LIN {X 0,Y 516.274,Z 395.585,A -85,B 0,C 180,E1 -4997.107,E2 -4997.107} C_VEL
LIN {X 0,Y 516.289,Z 396.844,A -85,B 0,C 180,E1 -4998.208,E2 -4998.208} C_VEL
LIN {X 0,Y 518.463,Z 408.41,A -85,B 0,C 180,E1 -4998.579,E2 -4998.579} C_VEL
LIN {X 0,Y 518.178,Z 420.619,A -85,B 0,C 180,E1 -4999.041,E2 -4999.041} C_VEL
LIN {X 0,Y 517.927,Z 432.987,A -85,B 0,C 180,E1 -4999.678,E2 -4999.678} C_VEL
LIN {X 0,Y 517.573,Z 444.529,A -85,B 0,C 180,E1 -5000.457,E2 -5000.457} C_VEL
LIN {X 0,Y 517.31,Z 455.837,A -85,B 0,C 180,E1 -5001.422,E2 -5001.422} C_VEL
LIN {X 0,Y 517.018,Z 465.136,A -85,B 0,C 180,E1 -5002.412,E2 -5002.412} C_VEL
LIN {X 0,Y 516.779,Z 473.686,A -85,B 0,C 180,E1 -5003.535,E2 -5003.535} C_VEL
LIN {X 0,Y 516.539,Z 480.957,A -85,B 0,C 180,E1 -5004.714,E2 -5004.714} C_VEL
LIN {X 0,Y 516.446,Z 486.584,A -85,B 0,C 180,E1 -5005.852,E2 -5005.852} C_VEL
LIN {X 0,Y 516.334,Z 491.147,A -85,B 0,C 180,E1 -5007.014,E2 -5007.014} C_VEL
LIN {X 0,Y 516.286,Z 495.193,A -85,B 0,C 180,E1 -5008.394,E2 -5008.394} C_VEL
LIN {X 0,Y 516.191,Z 497.831,A -85,B 0,C 180,E1 -5009.752,E2 -5009.752} C_VEL
LIN {X 0,Y 516.199,Z 498.912,A -85,B 0,C 180,E1 -5010.651,E2 -5010.651} C_VEL
LIN {X 0,Y 516.184,Z 499.461,A -85,B 0,C 180,E1 -5011.542,E2 -5011.542} C_VEL
LIN {X 0,Y 516.169,Z 499.49,A -85,B 0,C 180,E1 -5012.424,E2 -5012.424} C_VEL
LIN {X 0,Y 516.169,Z 499.058,A -85,B 0,C 180,E1 -5013.301,E2 -5013.301} C_VEL
LIN {X 0,Y 516.186,Z 498.084,A -85,B 0,C 180,E1 -5014.172,E2 -5014.172} C_VEL
LIN {X 0,Y 516.267,Z 496.647,A -85,B 0,C 180,E1 -5015.04,E2 -5015.04} C_VEL
LIN {X 0,Y 516.337,Z 493.561,A -85,B 0,C 180,E1 -5016.327,E2 -5016.327} C_VEL
LIN {X 0,Y 516.436,Z 488.822,A -85,B 0,C 180,E1 -5017.715,E2 -5017.715} C_VEL
LIN {X 0,Y 516.545,Z 482.626,A -85,B 0,C 180,E1 -5019.075,E2 -5019.075} C_VEL
LIN {X 0,Y 516.722,Z 475.326,A -85,B 0,C 180,E1 -5020.329,E2 -5020.329} C_VEL
LIN {X 0,Y 516.922,Z 467.803,A -85,B 0,C 180,E1 -5021.368,E2 -5021.368} C_VEL
LIN {X 0,Y 517.231,Z 458.063,A -85,B 0,C 180,E1 -5022.46,E2 -5022.46} C_VEL
LIN {X 0,Y 517.467,Z 448.555,A -85,B 0,C 180,E1 -5023.328,E2 -5023.328} C_VEL
LIN {X 0,Y 517.786,Z 437.368,A -85,B 0,C 180,E1 -5024.148,E2 -5024.148} C_VEL
LIN {X 0,Y 518.106,Z 425.293,A -85,B 0,C 180,E1 -5024.836,E2 -5024.836} C_VEL
LIN {X 0,Y 518.392,Z 412.692,A -85,B 0,C 180,E1 -5025.375,E2 -5025.375} C_VEL
LIN {X 0,Y 518.315,Z 407.593,A -85,B 0,C 180,E1 -5025.548,E2 -5025.548} C_VEL
LIN {X 0,Y 516.347,Z 397.146,A -85,B 0,C 180,E1 -5025.894,E2 -5025.894} C_VEL
LIN {X 0,Y 516.355,Z 393.731,A -85,B 0,C 180,E1 -5029.016,E2 -5029.016} C_VEL
LIN {X 0,Y 516.424,Z 390.407,A -85,B 0,C 180,E1 -5032.179,E2 -5032.179} C_VEL
LIN {X 0,Y 516.475,Z 387.929,A -85,B 0,C 180,E1 -5034.535,E2 -5034.535} C_VEL
LIN {X 0,Y 516.447,Z 385.452,A -85,B 0,C 180,E1 -5036.88,E2 -5036.88} C_VEL
LIN {X 0,Y 516.657,Z 382.989,A -85,B 0,C 180,E1 -5039.221,E2 -5039.221} C_VEL
LIN {X 0,Y 516.81,Z 381.331,A -85,B 0,C 180,E1 -5040.78,E2 -5040.78} C_VEL
LIN {X 0,Y 516.793,Z 377.272,A -85,B 0,C 180,E1 -5044.681,E2 -5044.681} C_VEL
LIN {X 0,Y 516.754,Z 376.473,A -85,B 0,C 180,E1 -5045.464,E2 -5045.464} C_VEL
LIN {X 0,Y 516.909,Z 376.103,A -85,B 0,C 180,E1 -5047.049,E2 -5047.049} C_VEL
LIN {X 0,Y 516.929,Z 376.095,A -85,B 0,C 180,E1 -5049.39,E2 -5049.39} C_VEL
LIN {X 0,Y 516.965,Z 376.093,A -85,B 0,C 180,E1 -5051.836,E2 -5051.836} C_VEL
LIN {X 0,Y 516.909,Z 376.097,A -85,B 0,C 180,E1 -5055.149,E2 -5055.149} C_VEL
LIN {X 0,Y 516.897,Z 376.098,A -85,B 0,C 180,E1 -5058.224,E2 -5058.224} C_VEL
LIN {X 0,Y 516.883,Z 376.103,A -85,B 0,C 180,E1 -5060.703,E2 -5060.703} C_VEL
LIN {X 0,Y 516.877,Z 376.1,A -85,B 0,C 180,E1 -5063.224,E2 -5063.224} C_VEL
LIN {X 0,Y 516.913,Z 376.096,A -85,B 0,C 180,E1 -5066.199,E2 -5066.199} C_VEL
LIN {X 0,Y 516.912,Z 376.098,A -85,B 0,C 180,E1 -5069.306,E2 -5069.306} C_VEL
LIN {X 0,Y 516.872,Z 376.104,A -85,B 0,C 180,E1 -5072.547,E2 -5072.547} C_VEL
LIN {X 0,Y 516.86,Z 376.106,A -85,B 0,C 180,E1 -5075.336,E2 -5075.336} C_VEL
LIN {X 0,Y 516.86,Z 376.103,A -85,B 0,C 180,E1 -5077.947,E2 -5077.947} C_VEL
LIN {X 0,Y 516.892,Z 376.1,A -85,B 0,C 180,E1 -5080.741,E2 -5080.741} C_VEL
LIN {X 0,Y 516.86,Z 376.104,A -85,B 0,C 180,E1 -5083.906,E2 -5083.906} C_VEL
LIN {X 0,Y 516.861,Z 376.105,A -85,B 0,C 180,E1 -5086.11,E2 -5086.11} C_VEL
LIN {X 0,Y 516.889,Z 376.104,A -85,B 0,C 180,E1 -5089.264,E2 -5089.264} C_VEL
LIN {X 0,Y 516.933,Z 376.22,A -85,B 0,C 180,E1 -5091.051,E2 -5091.051} C_VEL
LIN {X 0,Y 517.978,Z 382.454,A -85,B 0,C 180,E1 -5093.833,E2 -5093.833} C_VEL
LIN {X 0,Y 517.929,Z 387.606,A -85,B 0,C 180,E1 -5095.867,E2 -5095.867} C_VEL
LIN {X 0,Y 517.555,Z 395.985,A -85,B 0,C 180,E1 -5098.939,E2 -5098.939} C_VEL
LIN {X 0,Y 517.232,Z 404.927,A -85,B 0,C 180,E1 -5102.032,E2 -5102.032} C_VEL
LIN {X 0,Y 517.067,Z 414.228,A -85,B 0,C 180,E1 -5105.084,E2 -5105.084} C_VEL
LIN {X 0,Y 516.883,Z 423.643,A -85,B 0,C 180,E1 -5108.047,E2 -5108.047} C_VEL
LIN {X 0,Y 516.771,Z 431.808,A -85,B 0,C 180,E1 -5110.541,E2 -5110.541} C_VEL
LIN {X 0,Y 516.6,Z 441.466,A -85,B 0,C 180,E1 -5113.403,E2 -5113.403} C_VEL
LIN {X 0,Y 516.532,Z 450.706,A -85,B 0,C 180,E1 -5116.103,E2 -5116.103} C_VEL
LIN {X 0,Y 518.459,Z 463.813,A -85,B 0,C 180,E1 -5116.456,E2 -5116.456} C_VEL
LIN {X 0,Y 518.157,Z 476.925,A -85,B 0,C 180,E1 -5116.922,E2 -5116.922} C_VEL
LIN {X 0,Y 517.848,Z 489.403,A -85,B 0,C 180,E1 -5117.537,E2 -5117.537} C_VEL
LIN {X 0,Y 517.538,Z 500.606,A -85,B 0,C 180,E1 -5118.25,E2 -5118.25} C_VEL
LIN {X 0,Y 517.266,Z 511.613,A -85,B 0,C 180,E1 -5119.137,E2 -5119.137} C_VEL
LIN {X 0,Y 516.998,Z 520.585,A -85,B 0,C 180,E1 -5120.022,E2 -5120.022} C_VEL
LIN {X 0,Y 516.746,Z 530.339,A -85,B 0,C 180,E1 -5121.202,E2 -5121.202} C_VEL
LIN {X 0,Y 516.56,Z 538.106,A -85,B 0,C 180,E1 -5122.38,E2 -5122.38} C_VEL
LIN {X 0,Y 516.423,Z 545.262,A -85,B 0,C 180,E1 -5123.753,E2 -5123.753} C_VEL
LIN {X 0,Y 516.313,Z 550.022,A -85,B 0,C 180,E1 -5124.927,E2 -5124.927} C_VEL
LIN {X 0,Y 516.354,Z 553.665,A -85,B 0,C 180,E1 -5126.101,E2 -5126.101} C_VEL
LIN {X 0,Y 516.282,Z 555.538,A -85,B 0,C 180,E1 -5126.882,E2 -5126.882} C_VEL
LIN {X 0,Y 516.261,Z 556.944,A -85,B 0,C 180,E1 -5127.662,E2 -5127.662} C_VEL
LIN {X 0,Y 516.16,Z 558.554,A -85,B 0,C 180,E1 -5129.223,E2 -5129.223} C_VEL
LIN {X 0,Y 516.154,Z 558.771,A -85,B 0,C 180,E1 -5130.003,E2 -5130.003} C_VEL
LIN {X 0,Y 516.192,Z 557.944,A -85,B 0,C 180,E1 -5131.563,E2 -5131.563} C_VEL
LIN {X 0,Y 516.262,Z 556.945,A -85,B 0,C 180,E1 -5132.343,E2 -5132.343} C_VEL
LIN {X 0,Y 516.283,Z 555.54,A -85,B 0,C 180,E1 -5133.124,E2 -5133.124} C_VEL
LIN {X 0,Y 516.327,Z 552.586,A -85,B 0,C 180,E1 -5134.296,E2 -5134.296} C_VEL
LIN {X 0,Y 516.407,Z 548.586,A -85,B 0,C 180,E1 -5135.469,E2 -5135.469} C_VEL
LIN {X 0,Y 516.449,Z 543.248,A -85,B 0,C 180,E1 -5136.683,E2 -5136.683} C_VEL
LIN {X 0,Y 516.582,Z 536.95,A -85,B 0,C 180,E1 -5137.822,E2 -5137.822} C_VEL
LIN {X 0,Y 516.801,Z 528.869,A -85,B 0,C 180,E1 -5139,E2 -5139} C_VEL
LIN {X 0,Y 516.998,Z 520.632,A -85,B 0,C 180,E1 -5139.984,E2 -5139.984} C_VEL
LIN {X 0,Y 517.317,Z 510.597,A -85,B 0,C 180,E1 -5140.967,E2 -5140.967} C_VEL
LIN {X 0,Y 517.57,Z 500.686,A -85,B 0,C 180,E1 -5141.755,E2 -5141.755} C_VEL
LIN {X 0,Y 517.853,Z 489.517,A -85,B 0,C 180,E1 -5142.467,E2 -5142.467} C_VEL
LIN {X 0,Y 518.182,Z 476.997,A -85,B 0,C 180,E1 -5143.084,E2 -5143.084} C_VEL
LIN {X 0,Y 518.44,Z 463.848,A -85,B 0,C 180,E1 -5143.551,E2 -5143.551} C_VEL
LIN {X 0,Y 516.539,Z 450.746,A -85,B 0,C 180,E1 -5143.903,E2 -5143.903} C_VEL
LIN {X 0,Y 516.628,Z 441.751,A -85,B 0,C 180,E1 -5146.602,E2 -5146.602} C_VEL
LIN {X 0,Y 516.807,Z 432.31,A -85,B 0,C 180,E1 -5149.464,E2 -5149.464} C_VEL
LIN {X 0,Y 516.99,Z 421.628,A -85,B 0,C 180,E1 -5152.797,E2 -5152.797} C_VEL
LIN {X 0,Y 517.182,Z 412.366,A -85,B 0,C 180,E1 -5155.778,E2 -5155.778} C_VEL
LIN {X 0,Y 517.425,Z 403.177,A -85,B 0,C 180,E1 -5158.83,E2 -5158.83} C_VEL
LIN {X 0,Y 517.77,Z 394.07,A -85,B 0,C 180,E1 -5161.965,E2 -5161.965} C_VEL
LIN {X 0,Y 518.027,Z 387.92,A -85,B 0,C 180,E1 -5164.149,E2 -5164.149} C_VEL
LIN {X 0,Y 517.995,Z 382.478,A -85,B 0,C 180,E1 -5166.173,E2 -5166.173} C_VEL
LIN {X 0,Y 516.905,Z 376.101,A -85,B 0,C 180,E1 -5168.716,E2 -5168.716} C_VEL
LIN {X 0,Y 516.895,Z 376.102,A -85,B 0,C 180,E1 -5171.779,E2 -5171.779} C_VEL
LIN {X 0,Y 516.908,Z 376.096,A -85,B 0,C 180,E1 -5175.008,E2 -5175.008} C_VEL
LIN {X 0,Y 516.914,Z 376.098,A -85,B 0,C 180,E1 -5178.401,E2 -5178.401} C_VEL
LIN {X 0,Y 516.887,Z 376.103,A -85,B 0,C 180,E1 -5181.284,E2 -5181.284} C_VEL
LIN {X 0,Y 516.878,Z 376.102,A -85,B 0,C 180,E1 -5184.22,E2 -5184.22} C_VEL
LIN {X 0,Y 516.892,Z 376.1,A -85,B 0,C 180,E1 -5187.052,E2 -5187.052} C_VEL
LIN {X 0,Y 516.897,Z 376.098,A -85,B 0,C 180,E1 -5189.796,E2 -5189.796} C_VEL
LIN {X 0,Y 516.9,Z 376.098,A -85,B 0,C 180,E1 -5192.465,E2 -5192.465} C_VEL
LIN {X 0,Y 516.893,Z 376.1,A -85,B 0,C 180,E1 -5195.643,E2 -5195.643} C_VEL
LIN {X 0,Y 516.896,Z 376.099,A -85,B 0,C 180,E1 -5198.462,E2 -5198.462} C_VEL
LIN {X 0,Y 516.909,Z 376.098,A -85,B 0,C 180,E1 -5200.955,E2 -5200.955} C_VEL
LIN {X 0,Y 516.914,Z 376.096,A -85,B 0,C 180,E1 -5203.41,E2 -5203.41} C_VEL
LIN {X 0,Y 516.887,Z 376.099,A -85,B 0,C 180,E1 -5205.833,E2 -5205.833} C_VEL
LIN {X 0,Y 516.977,Z 376.091,A -85,B 0,C 180,E1 -5208.233,E2 -5208.233} C_VEL
LIN {X 0,Y 516.963,Z 376.09,A -85,B 0,C 180,E1 -5211.399,E2 -5211.399} C_VEL
LIN {X 0,Y 516.997,Z 376.086,A -85,B 0,C 180,E1 -5213.756,E2 -5213.756} C_VEL
LIN {X 0,Y 517.019,Z 376.084,A -85,B 0,C 180,E1 -5216.882,E2 -5216.882} C_VEL
LIN {X 0,Y 517.092,Z 376.076,A -85,B 0,C 180,E1 -5219.999,E2 -5219.999} C_VEL
LIN {X 0,Y 517.082,Z 376.075,A -85,B 0,C 180,E1 -5222.336,E2 -5222.336} C_VEL
LIN {X 0,Y 517.022,Z 376.085,A -85,B 0,C 180,E1 -5225.459,E2 -5225.459} C_VEL
LIN {X 0,Y 516.959,Z 376.092,A -85,B 0,C 180,E1 -5228.6,E2 -5228.6} C_VEL
LIN {X 0,Y 516.961,Z 376.09,A -85,B 0,C 180,E1 -5231.806,E2 -5231.806} C_VEL
LIN {X 0,Y 516.95,Z 376.093,A -85,B 0,C 180,E1 -5235.144,E2 -5235.144} C_VEL
LIN {X 0,Y 516.92,Z 376.095,A -85,B 0,C 180,E1 -5238.222,E2 -5238.222} C_VEL
LIN {X 0,Y 516.919,Z 376.097,A -85,B 0,C 180,E1 -5240.7,E2 -5240.7} C_VEL
LIN {X 0,Y 516.896,Z 376.099,A -85,B 0,C 180,E1 -5244.072,E2 -5244.072} C_VEL
LIN {X 0,Y 516.918,Z 376.097,A -85,B 0,C 180,E1 -5246.657,E2 -5246.657} C_VEL
LIN {X 0,Y 516.914,Z 376.098,A -85,B 0,C 180,E1 -5249.522,E2 -5249.522} C_VEL
LIN {X 0,Y 516.901,Z 376.1,A -85,B 0,C 180,E1 -5252.542,E2 -5252.542} C_VEL
LIN {X 0,Y 516.869,Z 376.102,A -85,B 0,C 180,E1 -5255.328,E2 -5255.328} C_VEL
LIN {X 0,Y 516.883,Z 376.102,A -85,B 0,C 180,E1 -5257.941,E2 -5257.941} C_VEL
LIN {X 0,Y 516.886,Z 376.101,A -85,B 0,C 180,E1 -5260.74,E2 -5260.74} C_VEL
LIN {X 0,Y 516.885,Z 376.099,A -85,B 0,C 180,E1 -5263.902,E2 -5263.902} C_VEL
LIN {X 0,Y 516.851,Z 376.104,A -85,B 0,C 180,E1 -5266.894,E2 -5266.894} C_VEL
LIN {X 0,Y 516.887,Z 376.101,A -85,B 0,C 180,E1 -5269.588,E2 -5269.588} C_VEL
LIN {X 0,Y 516.885,Z 376.101,A -85,B 0,C 180,E1 -5270.282,E2 -5270.282} C_VEL
LIN {X 0,Y 516.213,Z 376.186,A -85,B 0,C 180,E1 -5270.932,E2 -5270.932} C_VEL
LIN {X 0,Y 513.368,Z 376.541,A -85,B 0,C 180,E1 -5271.987,E2 -5271.987} C_VEL
LIN {X 0,Y 510.962,Z 376.842,A -85,B 0,C 180,E1 -5272.838,E2 -5272.838} C_VEL
LIN {X 0,Y 509.921,Z 376.969,A -85,B 0,C 180,E1 -5273.494,E2 -5273.494} C_VEL
LIN {X 0,Y 509.832,Z 376.979,A -85,B 0,C 180,E1 -5273.716,E2 -5273.716} C_VEL
LIN {X 0,Y 509.863,Z 376.978,A -85,B 0,C 180,E1 -5276.537,E2 -5276.537} C_VEL
LIN {X 0,Y 509.847,Z 376.978,A -85,B 0,C 180,E1 -5279.332,E2 -5279.332} C_VEL
LIN {X 0,Y 509.887,Z 376.974,A -85,B 0,C 180,E1 -5282.052,E2 -5282.052} C_VEL
LIN {X 0,Y 509.878,Z 376.974,A -85,B 0,C 180,E1 -5284.702,E2 -5284.702} C_VEL
LIN {X 0,Y 509.828,Z 376.981,A -85,B 0,C 180,E1 -5287.455,E2 -5287.455} C_VEL
LIN {X 0,Y 509.916,Z 376.97,A -85,B 0,C 180,E1 -5289.842,E2 -5289.842} C_VEL
LIN {X 0,Y 509.877,Z 376.971,A -85,B 0,C 180,E1 -5293.172,E2 -5293.172} C_VEL
LIN {X 0,Y 509.861,Z 376.976,A -85,B 0,C 180,E1 -5295.632,E2 -5295.632} C_VEL
LIN {X 0,Y 509.911,Z 376.97,A -85,B 0,C 180,E1 -5298.872,E2 -5298.872} C_VEL
LIN {X 0,Y 509.947,Z 376.967,A -85,B 0,C 180,E1 -5302.076,E2 -5302.076} C_VEL
LIN {X 0,Y 509.976,Z 376.963,A -85,B 0,C 180,E1 -5304.461,E2 -5304.461} C_VEL
LIN {X 0,Y 510.051,Z 376.953,A -85,B 0,C 180,E1 -5307.628,E2 -5307.628} C_VEL
LIN {X 0,Y 510.055,Z 376.951,A -85,B 0,C 180,E1 -5310.787,E2 -5310.787} C_VEL
LIN {X 0,Y 509.946,Z 376.964,A -85,B 0,C 180,E1 -5313.157,E2 -5313.157} C_VEL
LIN {X 0,Y 509.974,Z 376.962,A -85,B 0,C 180,E1 -5316.327,E2 -5316.327} C_VEL
LIN {X 0,Y 509.905,Z 376.969,A -85,B 0,C 180,E1 -5318.717,E2 -5318.717} C_VEL
LIN {X 0,Y 509.938,Z 376.967,A -85,B 0,C 180,E1 -5321.927,E2 -5321.927} C_VEL
LIN {X 0,Y 509.878,Z 376.973,A -85,B 0,C 180,E1 -5325.239,E2 -5325.239} C_VEL
LIN {X 0,Y 509.872,Z 376.974,A -85,B 0,C 180,E1 -5327.998,E2 -5327.998} C_VEL
LIN {X 0,Y 509.833,Z 376.978,A -85,B 0,C 180,E1 -5330.999,E2 -5330.999} C_VEL
LIN {X 0,Y 509.84,Z 376.977,A -85,B 0,C 180,E1 -5333.559,E2 -5333.559} C_VEL
LIN {X 0,Y 509.821,Z 376.981,A -85,B 0,C 180,E1 -5336.36,E2 -5336.36} C_VEL
LIN {X 0,Y 509.582,Z 377.013,A -85,B 0,C 180,E1 -5338.858,E2 -5338.858} C_VEL
LIN {X 0,Y 509.456,Z 377.033,A -85,B 0,C 180,E1 -5339.772,E2 -5339.772} C_VEL
LIN {X 0,Y 509.378,Z 380.119,A -85,B 0,C 180,E1 -5342.689,E2 -5342.689} C_VEL
LIN {X 0,Y 509.319,Z 383.194,A -85,B 0,C 180,E1 -5345.5,E2 -5345.5} C_VEL
LIN {X 0,Y 509.284,Z 386.378,A -85,B 0,C 180,E1 -5348.383,E2 -5348.383} C_VEL
LIN {X 0,Y 509.246,Z 389.82,A -85,B 0,C 180,E1 -5351.481,E2 -5351.481} C_VEL
LIN {X 0,Y 509.212,Z 393.462,A -85,B 0,C 180,E1 -5354.734,E2 -5354.734} C_VEL
LIN {X 0,Y 509.216,Z 397.177,A -85,B 0,C 180,E1 -5358.003,E2 -5358.003} C_VEL
LIN {X 0,Y 511.501,Z 409.221,A -85,B 0,C 180,E1 -5358.41,E2 -5358.41} C_VEL
LIN {X 0,Y 511.27,Z 422.157,A -85,B 0,C 180,E1 -5358.92,E2 -5358.92} C_VEL
LIN {X 0,Y 511.011,Z 433.292,A -85,B 0,C 180,E1 -5359.51,E2 -5359.51} C_VEL
LIN {X 0,Y 510.629,Z 445.146,A -85,B 0,C 180,E1 -5360.322,E2 -5360.322} C_VEL
LIN {X 0,Y 510.355,Z 455.392,A -85,B 0,C 180,E1 -5361.204,E2 -5361.204} C_VEL
LIN {X 0,Y 510.057,Z 464.675,A -85,B 0,C 180,E1 -5362.183,E2 -5362.183} C_VEL
LIN {X 0,Y 509.77,Z 473.618,A -85,B 0,C 180,E1 -5363.356,E2 -5363.356} C_VEL
LIN {X 0,Y 509.527,Z 481.237,A -85,B 0,C 180,E1 -5364.599,E2 -5364.599} C_VEL
LIN {X 0,Y 509.373,Z 487.418,A -85,B 0,C 180,E1 -5365.87,E2 -5365.87} C_VEL
LIN {X 0,Y 509.287,Z 491.531,A -85,B 0,C 180,E1 -5366.946,E2 -5366.946} C_VEL
LIN {X 0,Y 509.219,Z 495.639,A -85,B 0,C 180,E1 -5368.369,E2 -5368.369} C_VEL
LIN {X 0,Y 509.147,Z 497.527,A -85,B 0,C 180,E1 -5369.289,E2 -5369.289} C_VEL
LIN {X 0,Y 509.128,Z 499.087,A -85,B 0,C 180,E1 -5370.409,E2 -5370.409} C_VEL
LIN {X 0,Y 509.087,Z 499.965,A -85,B 0,C 180,E1 -5372.007,E2 -5372.007} C_VEL
LIN {X 0,Y 509.087,Z 499.72,A -85,B 0,C 180,E1 -5372.899,E2 -5372.899} C_VEL
LIN {X 0,Y 509.107,Z 498.999,A -85,B 0,C 180,E1 -5373.795,E2 -5373.795} C_VEL
LIN {X 0,Y 509.155,Z 497.809,A -85,B 0,C 180,E1 -5374.667,E2 -5374.667} C_VEL
LIN {X 0,Y 509.244,Z 494.958,A -85,B 0,C 180,E1 -5376.014,E2 -5376.014} C_VEL
LIN {X 0,Y 509.354,Z 491.143,A -85,B 0,C 180,E1 -5377.274,E2 -5377.274} C_VEL
LIN {X 0,Y 509.422,Z 486.001,A -85,B 0,C 180,E1 -5378.557,E2 -5378.557} C_VEL
LIN {X 0,Y 509.631,Z 479.445,A -85,B 0,C 180,E1 -5379.834,E2 -5379.834} C_VEL
LIN {X 0,Y 509.813,Z 472.712,A -85,B 0,C 180,E1 -5380.89,E2 -5380.89} C_VEL
LIN {X 0,Y 510.068,Z 463.686,A -85,B 0,C 180,E1 -5382.038,E2 -5382.038} C_VEL
LIN {X 0,Y 510.389,Z 453.425,A -85,B 0,C 180,E1 -5383.09,E2 -5383.09} C_VEL
LIN {X 0,Y 510.721,Z 443.332,A -85,B 0,C 180,E1 -5383.923,E2 -5383.923} C_VEL
LIN {X 0,Y 511.051,Z 432.035,A -85,B 0,C 180,E1 -5384.664,E2 -5384.664} C_VEL
LIN {X 0,Y 511.352,Z 420.106,A -85,B 0,C 180,E1 -5385.271,E2 -5385.271} C_VEL
LIN {X 0,Y 511.444,Z 408.72,A -85,B 0,C 180,E1 -5385.706,E2 -5385.706} C_VEL
LIN {X 0,Y 509.573,Z 399.17,A -85,B 0,C 180,E1 -5386.021,E2 -5386.021} C_VEL
LIN {X 0,Y 509.261,Z 397.636,A -85,B 0,C 180,E1 -5386.076,E2 -5386.076} C_VEL
LIN {X 0,Y 509.298,Z 394.628,A -85,B 0,C 180,E1 -5388.862,E2 -5388.862} C_VEL
LIN {X 0,Y 509.356,Z 391.228,A -85,B 0,C 180,E1 -5392.07,E2 -5392.07} C_VEL
LIN {X 0,Y 509.409,Z 388.715,A -85,B 0,C 180,E1 -5394.459,E2 -5394.459} C_VEL
LIN {X 0,Y 509.389,Z 386.246,A -85,B 0,C 180,E1 -5396.837,E2 -5396.837} C_VEL
LIN {X 0,Y 509.605,Z 383.758,A -85,B 0,C 180,E1 -5399.211,E2 -5399.211} C_VEL
LIN {X 0,Y 509.771,Z 382.109,A -85,B 0,C 180,E1 -5400.791,E2 -5400.791} C_VEL
LIN {X 0,Y 509.756,Z 378.043,A -85,B 0,C 180,E1 -5404.746,E2 -5404.746} C_VEL
LIN {X 0,Y 509.718,Z 377.23,A -85,B 0,C 180,E1 -5405.539,E2 -5405.539} C_VEL
LIN {X 0,Y 509.883,Z 376.974,A -85,B 0,C 180,E1 -5407.923,E2 -5407.923} C_VEL
LIN {X 0,Y 509.904,Z 376.969,A -85,B 0,C 180,E1 -5411.126,E2 -5411.126} C_VEL
LIN {X 0,Y 509.84,Z 376.979,A -85,B 0,C 180,E1 -5413.553,E2 -5413.553} C_VEL
LIN {X 0,Y 509.836,Z 376.979,A -85,B 0,C 180,E1 -5416.004,E2 -5416.004} C_VEL
LIN {X 0,Y 509.838,Z 376.977,A -85,B 0,C 180,E1 -5418.485,E2 -5418.485} C_VEL
LIN {X 0,Y 509.828,Z 376.98,A -85,B 0,C 180,E1 -5421.003,E2 -5421.003} C_VEL
LIN {X 0,Y 509.835,Z 376.981,A -85,B 0,C 180,E1 -5423.564,E2 -5423.564} C_VEL
LIN {X 0,Y 509.882,Z 376.973,A -85,B 0,C 180,E1 -5426.382,E2 -5426.382} C_VEL
LIN {X 0,Y 509.859,Z 376.974,A -85,B 0,C 180,E1 -5428.846,E2 -5428.846} C_VEL
LIN {X 0,Y 509.796,Z 376.983,A -85,B 0,C 180,E1 -5431.592,E2 -5431.592} C_VEL
LIN {X 0,Y 509.828,Z 376.98,A -85,B 0,C 180,E1 -5434.416,E2 -5434.416} C_VEL
LIN {X 0,Y 509.798,Z 376.984,A -85,B 0,C 180,E1 -5437.343,E2 -5437.343} C_VEL
LIN {X 0,Y 509.854,Z 376.977,A -85,B 0,C 180,E1 -5440.381,E2 -5440.381} C_VEL
LIN {X 0,Y 509.818,Z 376.983,A -85,B 0,C 180,E1 -5443.068,E2 -5443.068} C_VEL
LIN {X 0,Y 509.809,Z 376.984,A -85,B 0,C 180,E1 -5445.796,E2 -5445.796} C_VEL
LIN {X 0,Y 509.851,Z 376.981,A -85,B 0,C 180,E1 -5448.58,E2 -5448.58} C_VEL
LIN {X 0,Y 509.89,Z 377.177,A -85,B 0,C 180,E1 -5450.784,E2 -5450.784} C_VEL
LIN {X 0,Y 511.011,Z 383.665,A -85,B 0,C 180,E1 -5453.75,E2 -5453.75} C_VEL
LIN {X 0,Y 510.963,Z 388.44,A -85,B 0,C 180,E1 -5455.677,E2 -5455.677} C_VEL
LIN {X 0,Y 510.572,Z 396.168,A -85,B 0,C 180,E1 -5458.587,E2 -5458.587} C_VEL
LIN {X 0,Y 510.288,Z 402.199,A -85,B 0,C 180,E1 -5460.734,E2 -5460.734} C_VEL
LIN {X 0,Y 510.072,Z 410.541,A -85,B 0,C 180,E1 -5463.586,E2 -5463.586} C_VEL
LIN {X 0,Y 509.93,Z 417.93,A -85,B 0,C 180,E1 -5466.014,E2 -5466.014} C_VEL
LIN {X 0,Y 509.784,Z 425.981,A -85,B 0,C 180,E1 -5468.576,E2 -5468.576} C_VEL
LIN {X 0,Y 509.639,Z 435.527,A -85,B 0,C 180,E1 -5471.512,E2 -5471.512} C_VEL
LIN {X 0,Y 509.49,Z 446.814,A -85,B 0,C 180,E1 -5474.928,E2 -5474.928} C_VEL
LIN {X 0,Y 509.437,Z 450.07,A -85,B 0,C 180,E1 -5475.906,E2 -5475.906} C_VEL
LIN {X 0,Y 511.209,Z 462.286,A -85,B 0,C 180,E1 -5476.234,E2 -5476.234} C_VEL
LIN {X 0,Y 511.509,Z 465.634,A -85,B 0,C 180,E1 -5476.344,E2 -5476.344} C_VEL
LIN {X 0,Y 511.154,Z 478.614,A -85,B 0,C 180,E1 -5476.84,E2 -5476.84} C_VEL
LIN {X 0,Y 510.836,Z 490.57,A -85,B 0,C 180,E1 -5477.462,E2 -5477.462} C_VEL
LIN {X 0,Y 510.492,Z 501.404,A -85,B 0,C 180,E1 -5478.186,E2 -5478.186} C_VEL
LIN {X 0,Y 510.208,Z 512.174,A -85,B 0,C 180,E1 -5479.085,E2 -5479.085} C_VEL
LIN {X 0,Y 509.899,Z 521.886,A -85,B 0,C 180,E1 -5480.082,E2 -5480.082} C_VEL
LIN {X 0,Y 509.697,Z 529.857,A -85,B 0,C 180,E1 -5481.079,E2 -5481.079} C_VEL
LIN {X 0,Y 509.484,Z 537.64,A -85,B 0,C 180,E1 -5482.274,E2 -5482.274} C_VEL
LIN {X 0,Y 509.322,Z 544.81,A -85,B 0,C 180,E1 -5483.665,E2 -5483.665} C_VEL
LIN {X 0,Y 509.247,Z 549.585,A -85,B 0,C 180,E1 -5484.856,E2 -5484.856} C_VEL
LIN {X 0,Y 509.265,Z 553.236,A -85,B 0,C 180,E1 -5486.046,E2 -5486.046} C_VEL
LIN {X 0,Y 509.2,Z 555.117,A -85,B 0,C 180,E1 -5486.838,E2 -5486.838} C_VEL
LIN {X 0,Y 509.19,Z 556.528,A -85,B 0,C 180,E1 -5487.63,E2 -5487.63} C_VEL
LIN {X 0,Y 509.074,Z 558.144,A -85,B 0,C 180,E1 -5489.212,E2 -5489.212} C_VEL
LIN {X 0,Y 509.066,Z 558.366,A -85,B 0,C 180,E1 -5490.003,E2 -5490.003} C_VEL
LIN {X 0,Y 509.113,Z 557.54,A -85,B 0,C 180,E1 -5491.585,E2 -5491.585} C_VEL
LIN {X 0,Y 509.191,Z 556.543,A -85,B 0,C 180,E1 -5492.376,E2 -5492.376} C_VEL
LIN {X 0,Y 509.202,Z 555.137,A -85,B 0,C 180,E1 -5493.168,E2 -5493.168} C_VEL
LIN {X 0,Y 509.219,Z 552.18,A -85,B 0,C 180,E1 -5494.356,E2 -5494.356} C_VEL
LIN {X 0,Y 509.325,Z 548.179,A -85,B 0,C 180,E1 -5495.546,E2 -5495.546} C_VEL
LIN {X 0,Y 509.399,Z 542.473,A -85,B 0,C 180,E1 -5496.847,E2 -5496.847} C_VEL
LIN {X 0,Y 509.565,Z 535.288,A -85,B 0,C 180,E1 -5498.13,E2 -5498.13} C_VEL
LIN {X 0,Y 509.771,Z 526.943,A -85,B 0,C 180,E1 -5499.325,E2 -5499.325} C_VEL
LIN {X 0,Y 510.011,Z 518.381,A -85,B 0,C 180,E1 -5500.322,E2 -5500.322} C_VEL
LIN {X 0,Y 510.402,Z 507.817,A -85,B 0,C 180,E1 -5501.318,E2 -5501.318} C_VEL
LIN {X 0,Y 510.644,Z 496.78,A -85,B 0,C 180,E1 -5502.16,E2 -5502.16} C_VEL
LIN {X 0,Y 510.975,Z 485.924,A -85,B 0,C 180,E1 -5502.816,E2 -5502.816} C_VEL
LIN {X 0,Y 511.323,Z 474.144,A -85,B 0,C 180,E1 -5503.363,E2 -5503.363} C_VEL
LIN {X 0,Y 511.336,Z 462.885,A -85,B 0,C 180,E1 -5503.755,E2 -5503.755} C_VEL
LIN {X 0,Y 509.448,Z 450.372,A -85,B 0,C 180,E1 -5504.1,E2 -5504.1} C_VEL
LIN {X 0,Y 509.558,Z 441.399,A -85,B 0,C 180,E1 -5506.839,E2 -5506.839} C_VEL
LIN {X 0,Y 509.753,Z 432.028,A -85,B 0,C 180,E1 -5509.744,E2 -5509.744} C_VEL
LIN {X 0,Y 509.926,Z 422.74,A -85,B 0,C 180,E1 -5512.702,E2 -5512.702} C_VEL
LIN {X 0,Y 510.136,Z 413.505,A -85,B 0,C 180,E1 -5515.722,E2 -5515.722} C_VEL
LIN {X 0,Y 510.42,Z 404.333,A -85,B 0,C 180,E1 -5518.813,E2 -5518.813} C_VEL
LIN {X 0,Y 510.789,Z 395.229,A -85,B 0,C 180,E1 -5521.989,E2 -5521.989} C_VEL
LIN {X 0,Y 511.063,Z 388.564,A -85,B 0,C 180,E1 -5524.4,E2 -5524.4} C_VEL
LIN {X 0,Y 511.027,Z 383.66,A -85,B 0,C 180,E1 -5526.256,E2 -5526.256} C_VEL
LIN {X 0,Y 509.863,Z 376.977,A -85,B 0,C 180,E1 -5528.971,E2 -5528.971} C_VEL
LIN {X 0,Y 509.842,Z 376.98,A -85,B 0,C 180,E1 -5531.894,E2 -5531.894} C_VEL
LIN {X 0,Y 509.852,Z 376.978,A -85,B 0,C 180,E1 -5534.671,E2 -5534.671} C_VEL
LIN {X 0,Y 509.857,Z 376.975,A -85,B 0,C 180,E1 -5538.106,E2 -5538.106} C_VEL
LIN {X 0,Y 509.844,Z 376.977,A -85,B 0,C 180,E1 -5540.647,E2 -5540.647} C_VEL
LIN {X 0,Y 509.82,Z 376.982,A -85,B 0,C 180,E1 -5543.646,E2 -5543.646} C_VEL
LIN {X 0,Y 509.851,Z 376.977,A -85,B 0,C 180,E1 -5546.538,E2 -5546.538} C_VEL
LIN {X 0,Y 509.854,Z 376.979,A -85,B 0,C 180,E1 -5549.334,E2 -5549.334} C_VEL
LIN {X 0,Y 509.856,Z 376.977,A -85,B 0,C 180,E1 -5552.052,E2 -5552.052} C_VEL
LIN {X 0,Y 509.825,Z 376.982,A -85,B 0,C 180,E1 -5554.701,E2 -5554.701} C_VEL
LIN {X 0,Y 509.837,Z 376.98,A -85,B 0,C 180,E1 -5557.458,E2 -5557.458} C_VEL
LIN {X 0,Y 509.927,Z 376.969,A -85,B 0,C 180,E1 -5559.844,E2 -5559.844} C_VEL
LIN {X 0,Y 509.882,Z 376.973,A -85,B 0,C 180,E1 -5563.174,E2 -5563.174} C_VEL
LIN {X 0,Y 509.859,Z 376.975,A -85,B 0,C 180,E1 -5565.633,E2 -5565.633} C_VEL
LIN {X 0,Y 509.918,Z 376.968,A -85,B 0,C 180,E1 -5568.874,E2 -5568.874} C_VEL
LIN {X 0,Y 509.931,Z 376.968,A -85,B 0,C 180,E1 -5572.077,E2 -5572.077} C_VEL
LIN {X 0,Y 509.976,Z 376.961,A -85,B 0,C 180,E1 -5574.464,E2 -5574.464} C_VEL
LIN {X 0,Y 510.058,Z 376.951,A -85,B 0,C 180,E1 -5577.63,E2 -5577.63} C_VEL
LIN {X 0,Y 510.071,Z 376.949,A -85,B 0,C 180,E1 -5580.789,E2 -5580.789} C_VEL
LIN {X 0,Y 509.933,Z 376.967,A -85,B 0,C 180,E1 -5583.16,E2 -5583.16} C_VEL
LIN {X 0,Y 509.929,Z 376.966,A -85,B 0,C 180,E1 -5586.329,E2 -5586.329} C_VEL
LIN {X 0,Y 509.883,Z 376.974,A -85,B 0,C 180,E1 -5589.52,E2 -5589.52} C_VEL
LIN {X 0,Y 509.913,Z 376.969,A -85,B 0,C 180,E1 -5591.931,E2 -5591.931} C_VEL
LIN {X 0,Y 509.903,Z 376.97,A -85,B 0,C 180,E1 -5595.241,E2 -5595.241} C_VEL
LIN {X 0,Y 509.865,Z 376.975,A -85,B 0,C 180,E1 -5598.483,E2 -5598.483} C_VEL
LIN {X 0,Y 509.857,Z 376.976,A -85,B 0,C 180,E1 -5601.001,E2 -5601.001} C_VEL
LIN {X 0,Y 509.828,Z 376.978,A -85,B 0,C 180,E1 -5603.563,E2 -5603.563} C_VEL
LIN {X 0,Y 509.913,Z 376.969,A -85,B 0,C 180,E1 -5606.376,E2 -5606.376} C_VEL
LIN {X 0,Y 509.863,Z 376.976,A -85,B 0,C 180,E1 -5609.75,E2 -5609.75} C_VEL
LIN {X 0,Y 509.879,Z 376.973,A -85,B 0,C 180,E1 -5612.772,E2 -5612.772} C_VEL
LIN {X 0,Y 509.828,Z 376.978,A -85,B 0,C 180,E1 -5615.576,E2 -5615.576} C_VEL
LIN {X 0,Y 509.853,Z 376.976,A -85,B 0,C 180,E1 -5618.337,E2 -5618.337} C_VEL
LIN {X 0,Y 509.856,Z 376.977,A -85,B 0,C 180,E1 -5621.424,E2 -5621.424} C_VEL
LIN {X 0,Y 509.843,Z 376.979,A -85,B 0,C 180,E1 -5624.668,E2 -5624.668} C_VEL
LIN {X 0,Y 509.851,Z 376.976,A -85,B 0,C 180,E1 -5628.103,E2 -5628.103} C_VEL
LIN {X 0,Y 509.849,Z 376.977,A -85,B 0,C 180,E1 -5630.646,E2 -5630.646} C_VEL
LIN {X 0,Y 509.832,Z 376.979,A -85,B 0,C 180,E1 -5633.716,E2 -5633.716} C_VEL
LIN {X 0,Y 509.166,Z 377.062,A -85,B 0,C 180,E1 -5634.376,E2 -5634.376} C_VEL
LIN {X 0,Y 506.352,Z 377.413,A -85,B 0,C 180,E1 -5635.448,E2 -5635.448} C_VEL
LIN {X 0,Y 503.961,Z 377.712,A -85,B 0,C 180,E1 -5636.311,E2 -5636.311} C_VEL
LIN {X 0,Y 502.911,Z 377.84,A -85,B 0,C 180,E1 -5636.978,E2 -5636.978} C_VEL
LIN {X 0,Y 502.812,Z 377.852,A -85,B 0,C 180,E1 -5637.203,E2 -5637.203} C_VEL
LIN {X 0,Y 502.816,Z 377.853,A -85,B 0,C 180,E1 -5640.063,E2 -5640.063} C_VEL
LIN {X 0,Y 502.831,Z 377.851,A -85,B 0,C 180,E1 -5642.531,E2 -5642.531} C_VEL
LIN {X 0,Y 502.83,Z 377.85,A -85,B 0,C 180,E1 -5645.296,E2 -5645.296} C_VEL
LIN {X 0,Y 502.781,Z 377.857,A -85,B 0,C 180,E1 -5647.824,E2 -5647.824} C_VEL
LIN {X 0,Y 502.823,Z 377.852,A -85,B 0,C 180,E1 -5650.398,E2 -5650.398} C_VEL
LIN {X 0,Y 502.826,Z 377.851,A -85,B 0,C 180,E1 -5652.929,E2 -5652.929} C_VEL
LIN {X 0,Y 502.842,Z 377.851,A -85,B 0,C 180,E1 -5655.427,E2 -5655.427} C_VEL
LIN {X 0,Y 502.875,Z 377.845,A -85,B 0,C 180,E1 -5658.714,E2 -5658.714} C_VEL
LIN {X 0,Y 502.897,Z 377.845,A -85,B 0,C 180,E1 -5661.964,E2 -5661.964} C_VEL
LIN {X 0,Y 502.93,Z 377.84,A -85,B 0,C 180,E1 -5664.384,E2 -5664.384} C_VEL
LIN {X 0,Y 503.02,Z 377.829,A -85,B 0,C 180,E1 -5667.595,E2 -5667.595} C_VEL
LIN {X 0,Y 503.026,Z 377.826,A -85,B 0,C 180,E1 -5670.798,E2 -5670.798} C_VEL
LIN {X 0,Y 502.889,Z 377.843,A -85,B 0,C 180,E1 -5673.202,E2 -5673.202} C_VEL
LIN {X 0,Y 502.923,Z 377.841,A -85,B 0,C 180,E1 -5676.416,E2 -5676.416} C_VEL
LIN {X 0,Y 502.864,Z 377.846,A -85,B 0,C 180,E1 -5678.84,E2 -5678.84} C_VEL
LIN {X 0,Y 502.88,Z 377.848,A -85,B 0,C 180,E1 -5682.097,E2 -5682.097} C_VEL
LIN {X 0,Y 502.833,Z 377.85,A -85,B 0,C 180,E1 -5685.397,E2 -5685.397} C_VEL
LIN {X 0,Y 502.83,Z 377.851,A -85,B 0,C 180,E1 -5688.119,E2 -5688.119} C_VEL
LIN {X 0,Y 502.81,Z 377.853,A -85,B 0,C 180,E1 -5690.533,E2 -5690.533} C_VEL
LIN {X 0,Y 502.79,Z 377.857,A -85,B 0,C 180,E1 -5693.037,E2 -5693.037} C_VEL
LIN {X 0,Y 502.811,Z 377.856,A -85,B 0,C 180,E1 -5695.673,E2 -5695.673} C_VEL
LIN {X 0,Y 502.583,Z 377.885,A -85,B 0,C 180,E1 -5698.384,E2 -5698.384} C_VEL
LIN {X 0,Y 502.367,Z 378.13,A -85,B 0,C 180,E1 -5700.236,E2 -5700.236} C_VEL
LIN {X 0,Y 502.298,Z 381.183,A -85,B 0,C 180,E1 -5703.066,E2 -5703.066} C_VEL
LIN {X 0,Y 502.257,Z 384.354,A -85,B 0,C 180,E1 -5705.989,E2 -5705.989} C_VEL
LIN {X 0,Y 502.21,Z 387.703,A -85,B 0,C 180,E1 -5709.025,E2 -5709.025} C_VEL
LIN {X 0,Y 502.171,Z 391.206,A -85,B 0,C 180,E1 -5712.198,E2 -5712.198} C_VEL
LIN {X 0,Y 502.158,Z 393.737,A -85,B 0,C 180,E1 -5714.459,E2 -5714.459} C_VEL
LIN {X 0,Y 502.134,Z 397.543,A -85,B 0,C 180,E1 -5717.818,E2 -5717.818} C_VEL
LIN {X 0,Y 504.521,Z 409.336,A -85,B 0,C 180,E1 -5718.213,E2 -5718.213} C_VEL
LIN {X 0,Y 504.376,Z 422.689,A -85,B 0,C 180,E1 -5718.75,E2 -5718.75} C_VEL
LIN {X 0,Y 504.071,Z 434.437,A -85,B 0,C 180,E1 -5719.389,E2 -5719.389} C_VEL
LIN {X 0,Y 503.686,Z 445.9,A -85,B 0,C 180,E1 -5720.194,E2 -5720.194} C_VEL
LIN {X 0,Y 503.37,Z 455.981,A -85,B 0,C 180,E1 -5721.077,E2 -5721.077} C_VEL
LIN {X 0,Y 503.061,Z 465.23,A -85,B 0,C 180,E1 -5722.071,E2 -5722.071} C_VEL
LIN {X 0,Y 502.729,Z 474.412,A -85,B 0,C 180,E1 -5723.301,E2 -5723.301} C_VEL
LIN {X 0,Y 502.476,Z 482.179,A -85,B 0,C 180,E1 -5724.6,E2 -5724.6} C_VEL
LIN {X 0,Y 502.303,Z 488.534,A -85,B 0,C 180,E1 -5725.969,E2 -5725.969} C_VEL
LIN {X 0,Y 502.211,Z 492.635,A -85,B 0,C 180,E1 -5727.095,E2 -5727.095} C_VEL
LIN {X 0,Y 502.115,Z 496.696,A -85,B 0,C 180,E1 -5728.619,E2 -5728.619} C_VEL
LIN {X 0,Y 502.035,Z 499.316,A -85,B 0,C 180,E1 -5730.211,E2 -5730.211} C_VEL
LIN {X 0,Y 502.014,Z 500.343,A -85,B 0,C 180,E1 -5731.872,E2 -5731.872} C_VEL
LIN {X 0,Y 502.025,Z 499.832,A -85,B 0,C 180,E1 -5733.387,E2 -5733.387} C_VEL
LIN {X 0,Y 502.037,Z 498.835,A -85,B 0,C 180,E1 -5734.281,E2 -5734.281} C_VEL
LIN {X 0,Y 502.153,Z 496.792,A -85,B 0,C 180,E1 -5735.456,E2 -5735.456} C_VEL
LIN {X 0,Y 502.245,Z 492.92,A -85,B 0,C 180,E1 -5736.934,E2 -5736.934} C_VEL
LIN {X 0,Y 502.337,Z 488.194,A -85,B 0,C 180,E1 -5738.239,E2 -5738.239} C_VEL
LIN {X 0,Y 502.514,Z 482.017,A -85,B 0,C 180,E1 -5739.547,E2 -5739.547} C_VEL
LIN {X 0,Y 502.755,Z 474.374,A -85,B 0,C 180,E1 -5740.823,E2 -5740.823} C_VEL
LIN {X 0,Y 503.041,Z 466.248,A -85,B 0,C 180,E1 -5741.919,E2 -5741.919} C_VEL
LIN {X 0,Y 503.35,Z 456.867,A -85,B 0,C 180,E1 -5742.951,E2 -5742.951} C_VEL
LIN {X 0,Y 503.702,Z 445.621,A -85,B 0,C 180,E1 -5743.938,E2 -5743.938} C_VEL
LIN {X 0,Y 504.107,Z 434.024,A -85,B 0,C 180,E1 -5744.744,E2 -5744.744} C_VEL
LIN {X 0,Y 504.398,Z 422.251,A -85,B 0,C 180,E1 -5745.373,E2 -5745.373} C_VEL
LIN {X 0,Y 504.566,Z 409.866,A -85,B 0,C 180,E1 -5745.867,E2 -5745.867} C_VEL
LIN {X 0,Y 502.827,Z 400.939,A -85,B 0,C 180,E1 -5746.178,E2 -5746.178} C_VEL
LIN {X 0,Y 502.191,Z 398.132,A -85,B 0,C 180,E1 -5746.263,E2 -5746.263} C_VEL
LIN {X 0,Y 502.253,Z 395.506,A -85,B 0,C 180,E1 -5748.703,E2 -5748.703} C_VEL
LIN {X 0,Y 502.305,Z 392.058,A -85,B 0,C 180,E1 -5751.958,E2 -5751.958} C_VEL
LIN {X 0,Y 502.348,Z 389.538,A -85,B 0,C 180,E1 -5754.381,E2 -5754.381} C_VEL
LIN {X 0,Y 502.331,Z 387.039,A -85,B 0,C 180,E1 -5756.793,E2 -5756.793} C_VEL
LIN {X 0,Y 502.555,Z 384.551,A -85,B 0,C 180,E1 -5759.199,E2 -5759.199} C_VEL
LIN {X 0,Y 502.732,Z 382.888,A -85,B 0,C 180,E1 -5760.802,E2 -5760.802} C_VEL
LIN {X 0,Y 502.721,Z 378.806,A -85,B 0,C 180,E1 -5764.812,E2 -5764.812} C_VEL
LIN {X 0,Y 502.684,Z 378.015,A -85,B 0,C 180,E1 -5765.617,E2 -5765.617} C_VEL
LIN {X 0,Y 502.847,Z 377.851,A -85,B 0,C 180,E1 -5768.035,E2 -5768.035} C_VEL
LIN {X 0,Y 502.873,Z 377.846,A -85,B 0,C 180,E1 -5771.284,E2 -5771.284} C_VEL
LIN {X 0,Y 502.816,Z 377.854,A -85,B 0,C 180,E1 -5774.572,E2 -5774.572} C_VEL
LIN {X 0,Y 502.845,Z 377.85,A -85,B 0,C 180,E1 -5777.908,E2 -5777.908} C_VEL
LIN {X 0,Y 502.797,Z 377.858,A -85,B 0,C 180,E1 -5780.539,E2 -5780.539} C_VEL
LIN {X 0,Y 502.79,Z 377.854,A -85,B 0,C 180,E1 -5783.041,E2 -5783.041} C_VEL
LIN {X 0,Y 502.813,Z 377.852,A -85,B 0,C 180,E1 -5785.678,E2 -5785.678} C_VEL
LIN {X 0,Y 502.813,Z 377.854,A -85,B 0,C 180,E1 -5788.375,E2 -5788.375} C_VEL
LIN {X 0,Y 502.767,Z 377.859,A -85,B 0,C 180,E1 -5791.502,E2 -5791.502} C_VEL
LIN {X 0,Y 502.78,Z 377.858,A -85,B 0,C 180,E1 -5794.448,E2 -5794.448} C_VEL
LIN {X 0,Y 502.76,Z 377.862,A -85,B 0,C 180,E1 -5797.182,E2 -5797.182} C_VEL
LIN {X 0,Y 502.81,Z 377.856,A -85,B 0,C 180,E1 -5800.014,E2 -5800.014} C_VEL
LIN {X 0,Y 502.803,Z 377.855,A -85,B 0,C 180,E1 -5802.206,E2 -5802.206} C_VEL
LIN {X 0,Y 502.779,Z 377.859,A -85,B 0,C 180,E1 -5805.472,E2 -5805.472} C_VEL
LIN {X 0,Y 502.819,Z 377.855,A -85,B 0,C 180,E1 -5807.869,E2 -5807.869} C_VEL
LIN {X 0,Y 502.822,Z 377.966,A -85,B 0,C 180,E1 -5810.414,E2 -5810.414} C_VEL
LIN {X 0,Y 503.826,Z 383.718,A -85,B 0,C 180,E1 -5813.148,E2 -5813.148} C_VEL
LIN {X 0,Y 504.099,Z 387.212,A -85,B 0,C 180,E1 -5814.654,E2 -5814.654} C_VEL
LIN {X 0,Y 503.713,Z 394.462,A -85,B 0,C 180,E1 -5817.514,E2 -5817.514} C_VEL
LIN {X 0,Y 503.341,Z 402.139,A -85,B 0,C 180,E1 -5820.344,E2 -5820.344} C_VEL
LIN {X 0,Y 503.03,Z 411.034,A -85,B 0,C 180,E1 -5823.448,E2 -5823.448} C_VEL
LIN {X 0,Y 502.908,Z 417.714,A -85,B 0,C 180,E1 -5825.685,E2 -5825.685} C_VEL
LIN {X 0,Y 502.707,Z 426.96,A -85,B 0,C 180,E1 -5828.689,E2 -5828.689} C_VEL
LIN {X 0,Y 502.563,Z 435.07,A -85,B 0,C 180,E1 -5831.242,E2 -5831.242} C_VEL
LIN {X 0,Y 502.431,Z 445.946,A -85,B 0,C 180,E1 -5834.591,E2 -5834.591} C_VEL
LIN {X 0,Y 502.369,Z 449.583,A -85,B 0,C 180,E1 -5835.703,E2 -5835.703} C_VEL
LIN {X 0,Y 504.135,Z 462.229,A -85,B 0,C 180,E1 -5836.053,E2 -5836.053} C_VEL
LIN {X 0,Y 504.525,Z 466.559,A -85,B 0,C 180,E1 -5836.202,E2 -5836.202} C_VEL
LIN {X 0,Y 504.196,Z 479.161,A -85,B 0,C 180,E1 -5836.707,E2 -5836.707} C_VEL
LIN {X 0,Y 503.85,Z 490.117,A -85,B 0,C 180,E1 -5837.291,E2 -5837.291} C_VEL
LIN {X 0,Y 503.448,Z 502.173,A -85,B 0,C 180,E1 -5838.121,E2 -5838.121} C_VEL
LIN {X 0,Y 503.151,Z 512.739,A -85,B 0,C 180,E1 -5839.032,E2 -5839.032} C_VEL
LIN {X 0,Y 502.867,Z 521.387,A -85,B 0,C 180,E1 -5839.942,E2 -5839.942} C_VEL
LIN {X 0,Y 502.648,Z 529.374,A -85,B 0,C 180,E1 -5840.953,E2 -5840.953} C_VEL
LIN {X 0,Y 502.403,Z 537.174,A -85,B 0,C 180,E1 -5842.164,E2 -5842.164} C_VEL
LIN {X 0,Y 502.243,Z 543.903,A -85,B 0,C 180,E1 -5843.476,E2 -5843.476} C_VEL
LIN {X 0,Y 502.182,Z 549.149,A -85,B 0,C 180,E1 -5844.784,E2 -5844.784} C_VEL
LIN {X 0,Y 502.161,Z 552.808,A -85,B 0,C 180,E1 -5845.99,E2 -5845.99} C_VEL
LIN {X 0,Y 502.121,Z 554.697,A -85,B 0,C 180,E1 -5846.794,E2 -5846.794} C_VEL
LIN {X 0,Y 502.121,Z 556.112,A -85,B 0,C 180,E1 -5847.596,E2 -5847.596} C_VEL
LIN {X 0,Y 501.991,Z 557.736,A -85,B 0,C 180,E1 -5849.201,E2 -5849.201} C_VEL
LIN {X 0,Y 501.981,Z 557.96,A -85,B 0,C 180,E1 -5850.003,E2 -5850.003} C_VEL
LIN {X 0,Y 502.037,Z 557.137,A -85,B 0,C 180,E1 -5851.607,E2 -5851.607} C_VEL
LIN {X 0,Y 502.122,Z 556.142,A -85,B 0,C 180,E1 -5852.409,E2 -5852.409} C_VEL
LIN {X 0,Y 502.123,Z 554.734,A -85,B 0,C 180,E1 -5853.212,E2 -5853.212} C_VEL
LIN {X 0,Y 502.115,Z 551.774,A -85,B 0,C 180,E1 -5854.418,E2 -5854.418} C_VEL
LIN {X 0,Y 502.241,Z 547.771,A -85,B 0,C 180,E1 -5855.624,E2 -5855.624} C_VEL
LIN {X 0,Y 502.334,Z 541.704,A -85,B 0,C 180,E1 -5857.014,E2 -5857.014} C_VEL
LIN {X 0,Y 502.496,Z 534.867,A -85,B 0,C 180,E1 -5858.245,E2 -5858.245} C_VEL
LIN {X 0,Y 502.723,Z 526.517,A -85,B 0,C 180,E1 -5859.457,E2 -5859.457} C_VEL
LIN {X 0,Y 502.996,Z 517.945,A -85,B 0,C 180,E1 -5860.468,E2 -5860.468} C_VEL
LIN {X 0,Y 503.402,Z 507.371,A -85,B 0,C 180,E1 -5861.478,E2 -5861.478} C_VEL
LIN {X 0,Y 503.66,Z 495.747,A -85,B 0,C 180,E1 -5862.372,E2 -5862.372} C_VEL
LIN {X 0,Y 504.049,Z 483.489,A -85,B 0,C 180,E1 -5863.098,E2 -5863.098} C_VEL
LIN {X 0,Y 504.452,Z 471.08,A -85,B 0,C 180,E1 -5863.652,E2 -5863.652} C_VEL
LIN {X 0,Y 504.354,Z 463.308,A -85,B 0,C 180,E1 -5863.924,E2 -5863.924} C_VEL
LIN {X 0,Y 502.367,Z 449.998,A -85,B 0,C 180,E1 -5864.303,E2 -5864.303} C_VEL
LIN {X 0,Y 502.508,Z 441.086,A -85,B 0,C 180,E1 -5867.082,E2 -5867.082} C_VEL
LIN {X 0,Y 502.705,Z 431.773,A -85,B 0,C 180,E1 -5870.033,E2 -5870.033} C_VEL
LIN {X 0,Y 502.894,Z 422.513,A -85,B 0,C 180,E1 -5873.038,E2 -5873.038} C_VEL
LIN {X 0,Y 503.151,Z 413.303,A -85,B 0,C 180,E1 -5876.106,E2 -5876.106} C_VEL
LIN {X 0,Y 503.462,Z 404.178,A -85,B 0,C 180,E1 -5879.249,E2 -5879.249} C_VEL
LIN {X 0,Y 503.8,Z 396.382,A -85,B 0,C 180,E1 -5882.014,E2 -5882.014} C_VEL
LIN {X 0,Y 504.121,Z 388.673,A -85,B 0,C 180,E1 -5884.863,E2 -5884.863} C_VEL
LIN {X 0,Y 504.005,Z 384.685,A -85,B 0,C 180,E1 -5886.399,E2 -5886.399} C_VEL
LIN {X 0,Y 502.81,Z 377.856,A -85,B 0,C 180,E1 -5889.236,E2 -5889.236} C_VEL
LIN {X 0,Y 502.784,Z 377.858,A -85,B 0,C 180,E1 -5892.196,E2 -5892.196} C_VEL
LIN {X 0,Y 502.798,Z 377.854,A -85,B 0,C 180,E1 -5895.471,E2 -5895.471} C_VEL
LIN {X 0,Y 502.808,Z 377.853,A -85,B 0,C 180,E1 -5897.861,E2 -5897.861} C_VEL
LIN {X 0,Y 502.805,Z 377.855,A -85,B 0,C 180,E1 -5901.024,E2 -5901.024} C_VEL
LIN {X 0,Y 502.782,Z 377.858,A -85,B 0,C 180,E1 -5904.17,E2 -5904.17} C_VEL
LIN {X 0,Y 502.815,Z 377.854,A -85,B 0,C 180,E1 -5906.999,E2 -5906.999} C_VEL
LIN {X 0,Y 502.827,Z 377.85,A -85,B 0,C 180,E1 -5910.065,E2 -5910.065} C_VEL
LIN {X 0,Y 502.798,Z 377.855,A -85,B 0,C 180,E1 -5912.531,E2 -5912.531} C_VEL
LIN {X 0,Y 502.79,Z 377.856,A -85,B 0,C 180,E1 -5915.311,E2 -5915.311} C_VEL
LIN {X 0,Y 502.791,Z 377.854,A -85,B 0,C 180,E1 -5917.826,E2 -5917.826} C_VEL
LIN {X 0,Y 502.834,Z 377.851,A -85,B 0,C 180,E1 -5920.4,E2 -5920.4} C_VEL
LIN {X 0,Y 502.829,Z 377.853,A -85,B 0,C 180,E1 -5922.931,E2 -5922.931} C_VEL
LIN {X 0,Y 502.839,Z 377.852,A -85,B 0,C 180,E1 -5925.428,E2 -5925.428} C_VEL
LIN {X 0,Y 502.884,Z 377.844,A -85,B 0,C 180,E1 -5928.716,E2 -5928.716} C_VEL
LIN {X 0,Y 502.89,Z 377.844,A -85,B 0,C 180,E1 -5931.966,E2 -5931.966} C_VEL
LIN {X 0,Y 502.931,Z 377.838,A -85,B 0,C 180,E1 -5934.386,E2 -5934.386} C_VEL
LIN {X 0,Y 503.029,Z 377.827,A -85,B 0,C 180,E1 -5937.597,E2 -5937.597} C_VEL
LIN {X 0,Y 503.021,Z 377.827,A -85,B 0,C 180,E1 -5940.8,E2 -5940.8} C_VEL
LIN {X 0,Y 502.877,Z 377.845,A -85,B 0,C 180,E1 -5943.204,E2 -5943.204} C_VEL
LIN {X 0,Y 502.879,Z 377.845,A -85,B 0,C 180,E1 -5946.419,E2 -5946.419} C_VEL
LIN {X 0,Y 502.868,Z 377.846,A -85,B 0,C 180,E1 -5948.843,E2 -5948.843} C_VEL
LIN {X 0,Y 502.854,Z 377.849,A -85,B 0,C 180,E1 -5952.101,E2 -5952.101} C_VEL
LIN {X 0,Y 502.857,Z 377.847,A -85,B 0,C 180,E1 -5955.399,E2 -5955.399} C_VEL
LIN {X 0,Y 502.83,Z 377.853,A -85,B 0,C 180,E1 -5958.751,E2 -5958.751} C_VEL
LIN {X 0,Y 502.79,Z 377.857,A -85,B 0,C 180,E1 -5961.31,E2 -5961.31} C_VEL
LIN {X 0,Y 502.78,Z 377.856,A -85,B 0,C 180,E1 -5963.913,E2 -5963.913} C_VEL
LIN {X 0,Y 502.849,Z 377.849,A -85,B 0,C 180,E1 -5966.566,E2 -5966.566} C_VEL
LIN {X 0,Y 502.82,Z 377.854,A -85,B 0,C 180,E1 -5969.933,E2 -5969.933} C_VEL
LIN {X 0,Y 502.838,Z 377.85,A -85,B 0,C 180,E1 -5973.03,E2 -5973.03} C_VEL
LIN {X 0,Y 502.773,Z 377.857,A -85,B 0,C 180,E1 -5975.95,E2 -5975.95} C_VEL
LIN {X 0,Y 502.801,Z 377.857,A -85,B 0,C 180,E1 -5978.975,E2 -5978.975} C_VEL
LIN {X 0,Y 502.808,Z 377.854,A -85,B 0,C 180,E1 -5982.197,E2 -5982.197} C_VEL
LIN {X 0,Y 502.789,Z 377.857,A -85,B 0,C 180,E1 -5985.468,E2 -5985.468} C_VEL
LIN {X 0,Y 502.798,Z 377.854,A -85,B 0,C 180,E1 -5987.859,E2 -5987.859} C_VEL
LIN {X 0,Y 502.804,Z 377.856,A -85,B 0,C 180,E1 -5991.022,E2 -5991.022} C_VEL
LIN {X 0,Y 502.785,Z 377.858,A -85,B 0,C 180,E1 -5994.166,E2 -5994.166} C_VEL
LIN {X 0,Y 502.812,Z 377.852,A -85,B 0,C 180,E1 -5997.203,E2 -5997.203} C_VEL
LIN {X 0,Y 502.109,Z 377.943,A -85,B 0,C 180,E1 -5997.872,E2 -5997.872} C_VEL
LIN {X 0,Y 499.244,Z 378.3,A -85,B 0,C 180,E1 -5998.958,E2 -5998.958} C_VEL
LIN {X 0,Y 496.85,Z 378.597,A -85,B 0,C 180,E1 -5999.833,E2 -5999.833} C_VEL
LIN {X 0,Y 495.832,Z 378.726,A -85,B 0,C 180,E1 -6000.508,E2 -6000.508} C_VEL
LIN {X 0,Y 495.753,Z 378.73,A -85,B 0,C 180,E1 -6000.737,E2 -6000.737} C_VEL
LIN {X 0,Y 495.792,Z 378.727,A -85,B 0,C 180,E1 -6003.93,E2 -6003.93} C_VEL
LIN {X 0,Y 495.762,Z 378.733,A -85,B 0,C 180,E1 -6007.136,E2 -6007.136} C_VEL
LIN {X 0,Y 495.77,Z 378.732,A -85,B 0,C 180,E1 -6010.107,E2 -6010.107} C_VEL
LIN {X 0,Y 495.779,Z 378.73,A -85,B 0,C 180,E1 -6012.679,E2 -6012.679} C_VEL
LIN {X 0,Y 495.788,Z 378.729,A -85,B 0,C 180,E1 -6015.214,E2 -6015.214} C_VEL
LIN {X 0,Y 495.849,Z 378.721,A -85,B 0,C 180,E1 -6018.552,E2 -6018.552} C_VEL
LIN {X 0,Y 495.868,Z 378.719,A -85,B 0,C 180,E1 -6021.849,E2 -6021.849} C_VEL
LIN {X 0,Y 495.886,Z 378.717,A -85,B 0,C 180,E1 -6024.304,E2 -6024.304} C_VEL
LIN {X 0,Y 495.988,Z 378.705,A -85,B 0,C 180,E1 -6027.561,E2 -6027.561} C_VEL
LIN {X 0,Y 495.997,Z 378.702,A -85,B 0,C 180,E1 -6030.809,E2 -6030.809} C_VEL
LIN {X 0,Y 495.833,Z 378.721,A -85,B 0,C 180,E1 -6033.247,E2 -6033.247} C_VEL
LIN {X 0,Y 495.874,Z 378.72,A -85,B 0,C 180,E1 -6036.507,E2 -6036.507} C_VEL
LIN {X 0,Y 495.832,Z 378.723,A -85,B 0,C 180,E1 -6038.967,E2 -6038.967} C_VEL
LIN {X 0,Y 495.838,Z 378.723,A -85,B 0,C 180,E1 -6042.272,E2 -6042.272} C_VEL
LIN {X 0,Y 495.792,Z 378.727,A -85,B 0,C 180,E1 -6045.621,E2 -6045.621} C_VEL
LIN {X 0,Y 495.79,Z 378.728,A -85,B 0,C 180,E1 -6048.244,E2 -6048.244} C_VEL
LIN {X 0,Y 495.756,Z 378.731,A -85,B 0,C 180,E1 -6050.753,E2 -6050.753} C_VEL
LIN {X 0,Y 495.747,Z 378.733,A -85,B 0,C 180,E1 -6053.383,E2 -6053.383} C_VEL
LIN {X 0,Y 495.726,Z 378.736,A -85,B 0,C 180,E1 -6056.067,E2 -6056.067} C_VEL
LIN {X 0,Y 495.467,Z 378.771,A -85,B 0,C 180,E1 -6058.83,E2 -6058.83} C_VEL
LIN {X 0,Y 495.33,Z 378.793,A -85,B 0,C 180,E1 -6060.062,E2 -6060.062} C_VEL
LIN {X 0,Y 495.221,Z 381.921,A -85,B 0,C 180,E1 -6063.145,E2 -6063.145} C_VEL
LIN {X 0,Y 495.194,Z 385.021,A -85,B 0,C 180,E1 -6066.006,E2 -6066.006} C_VEL
LIN {X 0,Y 495.144,Z 387.942,A -85,B 0,C 180,E1 -6068.68,E2 -6068.68} C_VEL
LIN {X 0,Y 495.09,Z 390.723,A -85,B 0,C 180,E1 -6071.207,E2 -6071.207} C_VEL
LIN {X 0,Y 495.063,Z 393.897,A -85,B 0,C 180,E1 -6074.07,E2 -6074.07} C_VEL
LIN {X 0,Y 495.074,Z 397.237,A -85,B 0,C 180,E1 -6077.048,E2 -6077.048} C_VEL
LIN {X 0,Y 495.071,Z 397.974,A -85,B 0,C 180,E1 -6077.615,E2 -6077.615} C_VEL
LIN {X 0,Y 497.456,Z 409.406,A -85,B 0,C 180,E1 -6078.006,E2 -6078.006} C_VEL
LIN {X 0,Y 497.693,Z 415.381,A -85,B 0,C 180,E1 -6078.234,E2 -6078.234} C_VEL
LIN {X 0,Y 497.376,Z 427.467,A -85,B 0,C 180,E1 -6078.791,E2 -6078.791} C_VEL
LIN {X 0,Y 497.087,Z 438.116,A -85,B 0,C 180,E1 -6079.432,E2 -6079.432} C_VEL
LIN {X 0,Y 496.662,Z 448.585,A -85,B 0,C 180,E1 -6080.217,E2 -6080.217} C_VEL
LIN {X 0,Y 496.338,Z 458.48,A -85,B 0,C 180,E1 -6081.142,E2 -6081.142} C_VEL
LIN {X 0,Y 495.99,Z 467.763,A -85,B 0,C 180,E1 -6082.206,E2 -6082.206} C_VEL
LIN {X 0,Y 495.641,Z 476.559,A -85,B 0,C 180,E1 -6083.45,E2 -6083.45} C_VEL
LIN {X 0,Y 495.408,Z 483.502,A -85,B 0,C 180,E1 -6084.685,E2 -6084.685} C_VEL
LIN {X 0,Y 495.238,Z 489.006,A -85,B 0,C 180,E1 -6085.907,E2 -6085.907} C_VEL
LIN {X 0,Y 495.107,Z 494.032,A -85,B 0,C 180,E1 -6087.358,E2 -6087.358} C_VEL
LIN {X 0,Y 495.049,Z 496.711,A -85,B 0,C 180,E1 -6088.399,E2 -6088.399} C_VEL
LIN {X 0,Y 494.956,Z 499.511,A -85,B 0,C 180,E1 -6090.005,E2 -6090.005} C_VEL
LIN {X 0,Y 494.926,Z 500.709,A -85,B 0,C 180,E1 -6091.682,E2 -6091.682} C_VEL
LIN {X 0,Y 494.933,Z 500.204,A -85,B 0,C 180,E1 -6093.446,E2 -6093.446} C_VEL
LIN {X 0,Y 495.054,Z 497.646,A -85,B 0,C 180,E1 -6095.298,E2 -6095.298} C_VEL
LIN {X 0,Y 495.147,Z 494.588,A -85,B 0,C 180,E1 -6096.584,E2 -6096.584} C_VEL
LIN {X 0,Y 495.271,Z 490.216,A -85,B 0,C 180,E1 -6097.912,E2 -6097.912} C_VEL
LIN {X 0,Y 495.399,Z 484.553,A -85,B 0,C 180,E1 -6099.228,E2 -6099.228} C_VEL
LIN {X 0,Y 495.628,Z 477.409,A -85,B 0,C 180,E1 -6100.536,E2 -6100.536} C_VEL
LIN {X 0,Y 495.92,Z 469.48,A -85,B 0,C 180,E1 -6101.699,E2 -6101.699} C_VEL
LIN {X 0,Y 496.292,Z 460.097,A -85,B 0,C 180,E1 -6102.807,E2 -6102.807} C_VEL
LIN {X 0,Y 496.65,Z 449.497,A -85,B 0,C 180,E1 -6103.82,E2 -6103.82} C_VEL
LIN {X 0,Y 496.998,Z 438.96,A -85,B 0,C 180,E1 -6104.625,E2 -6104.625} C_VEL
LIN {X 0,Y 497.407,Z 426.409,A -85,B 0,C 180,E1 -6105.372,E2 -6105.372} C_VEL
LIN {X 0,Y 497.729,Z 414.548,A -85,B 0,C 180,E1 -6105.903,E2 -6105.903} C_VEL
LIN {X 0,Y 497.542,Z 409.782,A -85,B 0,C 180,E1 -6106.08,E2 -6106.08} C_VEL
LIN {X 0,Y 495.404,Z 400.038,A -85,B 0,C 180,E1 -6106.425,E2 -6106.425} C_VEL
LIN {X 0,Y 495.117,Z 398.579,A -85,B 0,C 180,E1 -6106.482,E2 -6106.482} C_VEL
LIN {X 0,Y 495.209,Z 396.372,A -85,B 0,C 180,E1 -6108.541,E2 -6108.541} C_VEL
LIN {X 0,Y 495.236,Z 392.897,A -85,B 0,C 180,E1 -6111.842,E2 -6111.842} C_VEL
LIN {X 0,Y 495.29,Z 390.376,A -85,B 0,C 180,E1 -6114.3,E2 -6114.3} C_VEL
LIN {X 0,Y 495.275,Z 387.852,A -85,B 0,C 180,E1 -6116.747,E2 -6116.747} C_VEL
LIN {X 0,Y 495.505,Z 385.345,A -85,B 0,C 180,E1 -6119.188,E2 -6119.188} C_VEL
LIN {X 0,Y 495.694,Z 383.701,A -85,B 0,C 180,E1 -6120.813,E2 -6120.813} C_VEL
LIN {X 0,Y 495.687,Z 379.623,A -85,B 0,C 180,E1 -6124.881,E2 -6124.881} C_VEL
LIN {X 0,Y 495.653,Z 378.81,A -85,B 0,C 180,E1 -6125.697,E2 -6125.697} C_VEL
LIN {X 0,Y 495.806,Z 378.728,A -85,B 0,C 180,E1 -6128.15,E2 -6128.15} C_VEL
LIN {X 0,Y 495.844,Z 378.722,A -85,B 0,C 180,E1 -6131.446,E2 -6131.446} C_VEL
LIN {X 0,Y 495.759,Z 378.735,A -85,B 0,C 180,E1 -6134.784,E2 -6134.784} C_VEL
LIN {X 0,Y 495.798,Z 378.727,A -85,B 0,C 180,E1 -6138.172,E2 -6138.172} C_VEL
LIN {X 0,Y 495.743,Z 378.736,A -85,B 0,C 180,E1 -6140.758,E2 -6140.758} C_VEL
LIN {X 0,Y 495.743,Z 378.734,A -85,B 0,C 180,E1 -6143.388,E2 -6143.388} C_VEL
LIN {X 0,Y 495.769,Z 378.73,A -85,B 0,C 180,E1 -6146.07,E2 -6146.07} C_VEL
LIN {X 0,Y 495.751,Z 378.732,A -85,B 0,C 180,E1 -6148.817,E2 -6148.817} C_VEL
LIN {X 0,Y 495.729,Z 378.735,A -85,B 0,C 180,E1 -6151.729,E2 -6151.729} C_VEL
LIN {X 0,Y 495.75,Z 378.733,A -85,B 0,C 180,E1 -6154.699,E2 -6154.699} C_VEL
LIN {X 0,Y 495.71,Z 378.738,A -85,B 0,C 180,E1 -6157.564,E2 -6157.564} C_VEL
LIN {X 0,Y 495.762,Z 378.732,A -85,B 0,C 180,E1 -6160.701,E2 -6160.701} C_VEL
LIN {X 0,Y 495.712,Z 378.738,A -85,B 0,C 180,E1 -6163.699,E2 -6163.699} C_VEL
LIN {X 0,Y 495.714,Z 378.739,A -85,B 0,C 180,E1 -6166.308,E2 -6166.308} C_VEL
LIN {X 0,Y 495.763,Z 378.737,A -85,B 0,C 180,E1 -6169.305,E2 -6169.305} C_VEL
LIN {X 0,Y 495.8,Z 378.854,A -85,B 0,C 180,E1 -6170.093,E2 -6170.093} C_VEL
LIN {X 0,Y 496.844,Z 384.928,A -85,B 0,C 180,E1 -6173.051,E2 -6173.051} C_VEL
LIN {X 0,Y 497.143,Z 388.428,A -85,B 0,C 180,E1 -6174.582,E2 -6174.582} C_VEL
LIN {X 0,Y 496.735,Z 395.651,A -85,B 0,C 180,E1 -6177.482,E2 -6177.482} C_VEL
LIN {X 0,Y 496.321,Z 403.108,A -85,B 0,C 180,E1 -6180.295,E2 -6180.295} C_VEL
LIN {X 0,Y 496.005,Z 411.274,A -85,B 0,C 180,E1 -6183.21,E2 -6183.21} C_VEL
LIN {X 0,Y 495.838,Z 418.662,A -85,B 0,C 180,E1 -6185.734,E2 -6185.734} C_VEL
LIN {X 0,Y 495.66,Z 426.627,A -85,B 0,C 180,E1 -6188.371,E2 -6188.371} C_VEL
LIN {X 0,Y 495.503,Z 434.67,A -85,B 0,C 180,E1 -6190.964,E2 -6190.964} C_VEL
LIN {X 0,Y 495.351,Z 445.47,A -85,B 0,C 180,E1 -6194.365,E2 -6194.365} C_VEL
LIN {X 0,Y 495.298,Z 449.11,A -85,B 0,C 180,E1 -6195.495,E2 -6195.495} C_VEL
LIN {X 0,Y 497.157,Z 462.847,A -85,B 0,C 180,E1 -6195.889,E2 -6195.889} C_VEL
LIN {X 0,Y 497.6,Z 467.467,A -85,B 0,C 180,E1 -6196.059,E2 -6196.059} C_VEL
LIN {X 0,Y 497.244,Z 479.671,A -85,B 0,C 180,E1 -6196.569,E2 -6196.569} C_VEL
LIN {X 0,Y 496.862,Z 490.231,A -85,B 0,C 180,E1 -6197.152,E2 -6197.152} C_VEL
LIN {X 0,Y 496.456,Z 501.64,A -85,B 0,C 180,E1 -6197.951,E2 -6197.951} C_VEL
LIN {X 0,Y 496.154,Z 512.225,A -85,B 0,C 180,E1 -6198.876,E2 -6198.876} C_VEL
LIN {X 0,Y 495.829,Z 520.888,A -85,B 0,C 180,E1 -6199.798,E2 -6199.798} C_VEL
LIN {X 0,Y 495.576,Z 528.889,A -85,B 0,C 180,E1 -6200.823,E2 -6200.823} C_VEL
LIN {X 0,Y 495.342,Z 536.709,A -85,B 0,C 180,E1 -6202.052,E2 -6202.052} C_VEL
LIN {X 0,Y 495.162,Z 543.912,A -85,B 0,C 180,E1 -6203.483,E2 -6203.483} C_VEL
LIN {X 0,Y 495.117,Z 548.713,A -85,B 0,C 180,E1 -6204.709,E2 -6204.709} C_VEL
LIN {X 0,Y 495.056,Z 552.38,A -85,B 0,C 180,E1 -6205.933,E2 -6205.933} C_VEL
LIN {X 0,Y 495.044,Z 554.276,A -85,B 0,C 180,E1 -6206.748,E2 -6206.748} C_VEL
LIN {X 0,Y 495.054,Z 555.697,A -85,B 0,C 180,E1 -6207.562,E2 -6207.562} C_VEL
LIN {X 0,Y 494.911,Z 557.329,A -85,B 0,C 180,E1 -6209.189,E2 -6209.189} C_VEL
LIN {X 0,Y 494.899,Z 557.554,A -85,B 0,C 180,E1 -6210.003,E2 -6210.003} C_VEL
LIN {X 0,Y 494.964,Z 556.735,A -85,B 0,C 180,E1 -6211.63,E2 -6211.63} C_VEL
LIN {X 0,Y 495.055,Z 555.741,A -85,B 0,C 180,E1 -6212.444,E2 -6212.444} C_VEL
LIN {X 0,Y 495.045,Z 554.332,A -85,B 0,C 180,E1 -6213.258,E2 -6213.258} C_VEL
LIN {X 0,Y 495.019,Z 551.369,A -85,B 0,C 180,E1 -6214.481,E2 -6214.481} C_VEL
LIN {X 0,Y 495.157,Z 547.364,A -85,B 0,C 180,E1 -6215.705,E2 -6215.705} C_VEL
LIN {X 0,Y 495.26,Z 541.188,A -85,B 0,C 180,E1 -6217.135,E2 -6217.135} C_VEL
LIN {X 0,Y 495.441,Z 534.448,A -85,B 0,C 180,E1 -6218.363,E2 -6218.363} C_VEL
LIN {X 0,Y 495.679,Z 526.09,A -85,B 0,C 180,E1 -6219.593,E2 -6219.593} C_VEL
LIN {X 0,Y 495.993,Z 517.509,A -85,B 0,C 180,E1 -6220.617,E2 -6220.617} C_VEL
LIN {X 0,Y 496.408,Z 506.927,A -85,B 0,C 180,E1 -6221.642,E2 -6221.642} C_VEL
LIN {X 0,Y 496.653,Z 496.381,A -85,B 0,C 180,E1 -6222.471,E2 -6222.471} C_VEL
LIN {X 0,Y 497.075,Z 485.001,A -85,B 0,C 180,E1 -6223.181,E2 -6223.181} C_VEL
LIN {X 0,Y 497.515,Z 471.895,A -85,B 0,C 180,E1 -6223.794,E2 -6223.794} C_VEL
LIN {X 0,Y 497.417,Z 464.086,A -85,B 0,C 180,E1 -6224.083,E2 -6224.083} C_VEL
LIN {X 0,Y 495.516,Z 451.38,A -85,B 0,C 180,E1 -6224.464,E2 -6224.464} C_VEL
LIN {X 0,Y 495.293,Z 449.574,A -85,B 0,C 180,E1 -6224.538,E2 -6224.538} C_VEL
LIN {X 0,Y 495.447,Z 440.772,A -85,B 0,C 180,E1 -6227.333,E2 -6227.333} C_VEL
LIN {X 0,Y 495.647,Z 431.704,A -85,B 0,C 180,E1 -6230.269,E2 -6230.269} C_VEL
LIN {X 0,Y 495.874,Z 422.293,A -85,B 0,C 180,E1 -6233.383,E2 -6233.383} C_VEL
LIN {X 0,Y 496.123,Z 413.305,A -85,B 0,C 180,E1 -6236.437,E2 -6236.437} C_VEL
LIN {X 0,Y 496.452,Z 405.297,A -85,B 0,C 180,E1 -6239.238,E2 -6239.238} C_VEL
LIN {X 0,Y 496.812,Z 396.251,A -85,B 0,C 180,E1 -6242.52,E2 -6242.52} C_VEL
LIN {X 0,Y 497.154,Z 389.826,A -85,B 0,C 180,E1 -6244.923,E2 -6244.923} C_VEL
LIN {X 0,Y 497.04,Z 385.981,A -85,B 0,C 180,E1 -6246.434,E2 -6246.434} C_VEL
LIN {X 0,Y 495.756,Z 378.734,A -85,B 0,C 180,E1 -6249.528,E2 -6249.528} C_VEL
LIN {X 0,Y 495.725,Z 378.736,A -85,B 0,C 180,E1 -6252.505,E2 -6252.505} C_VEL
LIN {X 0,Y 495.75,Z 378.732,A -85,B 0,C 180,E1 -6255.142,E2 -6255.142} C_VEL
LIN {X 0,Y 495.757,Z 378.732,A -85,B 0,C 180,E1 -6258.218,E2 -6258.218} C_VEL
LIN {X 0,Y 495.757,Z 378.734,A -85,B 0,C 180,E1 -6261.408,E2 -6261.408} C_VEL
LIN {X 0,Y 495.755,Z 378.732,A -85,B 0,C 180,E1 -6264.462,E2 -6264.462} C_VEL
LIN {X 0,Y 495.764,Z 378.731,A -85,B 0,C 180,E1 -6267.405,E2 -6267.405} C_VEL
LIN {X 0,Y 495.775,Z 378.729,A -85,B 0,C 180,E1 -6270.254,E2 -6270.254} C_VEL
LIN {X 0,Y 495.753,Z 378.736,A -85,B 0,C 180,E1 -6273.27,E2 -6273.27} C_VEL
LIN {X 0,Y 495.731,Z 378.737,A -85,B 0,C 180,E1 -6275.723,E2 -6275.723} C_VEL
LIN {X 0,Y 495.752,Z 378.732,A -85,B 0,C 180,E1 -6278.371,E2 -6278.371} C_VEL
LIN {X 0,Y 495.792,Z 378.728,A -85,B 0,C 180,E1 -6280.971,E2 -6280.971} C_VEL
LIN {X 0,Y 495.819,Z 378.726,A -85,B 0,C 180,E1 -6284.376,E2 -6284.376} C_VEL
LIN {X 0,Y 495.799,Z 378.728,A -85,B 0,C 180,E1 -6287.723,E2 -6287.723} C_VEL
LIN {X 0,Y 495.794,Z 378.726,A -85,B 0,C 180,E1 -6290.206,E2 -6290.206} C_VEL
LIN {X 0,Y 495.923,Z 378.712,A -85,B 0,C 180,E1 -6292.761,E2 -6292.761} C_VEL
LIN {X 0,Y 495.841,Z 378.722,A -85,B 0,C 180,E1 -6295.121,E2 -6295.121} C_VEL
LIN {X 0,Y 495.998,Z 378.703,A -85,B 0,C 180,E1 -6297.563,E2 -6297.563} C_VEL
LIN {X 0,Y 495.972,Z 378.705,A -85,B 0,C 180,E1 -6300.811,E2 -6300.811} C_VEL
LIN {X 0,Y 495.991,Z 378.703,A -85,B 0,C 180,E1 -6302.436,E2 -6302.436} C_VEL
LIN {X 0,Y 495.88,Z 378.717,A -85,B 0,C 180,E1 -6305.693,E2 -6305.693} C_VEL
LIN {X 0,Y 495.838,Z 378.722,A -85,B 0,C 180,E1 -6308.969,E2 -6308.969} C_VEL
LIN {X 0,Y 495.837,Z 378.722,A -85,B 0,C 180,E1 -6312.033,E2 -6312.033} C_VEL
LIN {X 0,Y 495.832,Z 378.721,A -85,B 0,C 180,E1 -6315.45,E2 -6315.45} C_VEL
LIN {X 0,Y 495.786,Z 378.73,A -85,B 0,C 180,E1 -6319.027,E2 -6319.027} C_VEL
LIN {X 0,Y 495.749,Z 378.734,A -85,B 0,C 180,E1 -6321.628,E2 -6321.628} C_VEL
LIN {X 0,Y 495.757,Z 378.732,A -85,B 0,C 180,E1 -6324.864,E2 -6324.864} C_VEL
LIN {X 0,Y 495.785,Z 378.731,A -85,B 0,C 180,E1 -6326.975,E2 -6326.975} C_VEL
LIN {X 0,Y 495.77,Z 378.731,A -85,B 0,C 180,E1 -6330.145,E2 -6330.145} C_VEL
LIN {X 0,Y 495.799,Z 378.727,A -85,B 0,C 180,E1 -6333.243,E2 -6333.243} C_VEL
LIN {X 0,Y 495.717,Z 378.737,A -85,B 0,C 180,E1 -6336.085,E2 -6336.085} C_VEL
LIN {X 0,Y 495.765,Z 378.733,A -85,B 0,C 180,E1 -6338.766,E2 -6338.766} C_VEL
LIN {X 0,Y 495.755,Z 378.733,A -85,B 0,C 180,E1 -6341.78,E2 -6341.78} C_VEL
LIN {X 0,Y 495.741,Z 378.734,A -85,B 0,C 180,E1 -6345.139,E2 -6345.139} C_VEL
LIN {X 0,Y 495.754,Z 378.733,A -85,B 0,C 180,E1 -6348.216,E2 -6348.216} C_VEL
LIN {X 0,Y 495.753,Z 378.733,A -85,B 0,C 180,E1 -6351.406,E2 -6351.406} C_VEL
LIN {X 0,Y 495.758,Z 378.732,A -85,B 0,C 180,E1 -6354.461,E2 -6354.461} C_VEL
LIN {X 0,Y 495.77,Z 378.73,A -85,B 0,C 180,E1 -6357.403,E2 -6357.403} C_VEL
LIN {X 0,Y 495.753,Z 378.73,A -85,B 0,C 180,E1 -6360.737,E2 -6360.737} C_VEL
LIN {X 0,Y 495.094,Z 378.814,A -85,B 0,C 180,E1 -6361.416,E2 -6361.416} C_VEL
LIN {X 0,Y 492.238,Z 379.171,A -85,B 0,C 180,E1 -6362.519,E2 -6362.519} C_VEL
LIN {X 0,Y 489.831,Z 379.471,A -85,B 0,C 180,E1 -6363.407,E2 -6363.407} C_VEL
LIN {X 0,Y 488.816,Z 379.597,A -85,B 0,C 180,E1 -6364.094,E2 -6364.094} C_VEL
LIN {X 0,Y 488.743,Z 379.607,A -85,B 0,C 180,E1 -6364.326,E2 -6364.326} C_VEL
LIN {X 0,Y 488.725,Z 379.609,A -85,B 0,C 180,E1 -6367.151,E2 -6367.151} C_VEL
LIN {X 0,Y 488.724,Z 379.609,A -85,B 0,C 180,E1 -6369.808,E2 -6369.808} C_VEL
LIN {X 0,Y 488.727,Z 379.61,A -85,B 0,C 180,E1 -6372.421,E2 -6372.421} C_VEL
LIN {X 0,Y 488.76,Z 379.605,A -85,B 0,C 180,E1 -6374.997,E2 -6374.997} C_VEL
LIN {X 0,Y 488.803,Z 379.599,A -85,B 0,C 180,E1 -6378.385,E2 -6378.385} C_VEL
LIN {X 0,Y 488.813,Z 379.597,A -85,B 0,C 180,E1 -6381.731,E2 -6381.731} C_VEL
LIN {X 0,Y 488.844,Z 379.594,A -85,B 0,C 180,E1 -6384.221,E2 -6384.221} C_VEL
LIN {X 0,Y 488.956,Z 379.581,A -85,B 0,C 180,E1 -6387.526,E2 -6387.526} C_VEL
LIN {X 0,Y 488.946,Z 379.58,A -85,B 0,C 180,E1 -6390.821,E2 -6390.821} C_VEL
LIN {X 0,Y 488.954,Z 379.582,A -85,B 0,C 180,E1 -6392.468,E2 -6392.468} C_VEL
LIN {X 0,Y 488.849,Z 379.593,A -85,B 0,C 180,E1 -6395.773,E2 -6395.773} C_VEL
LIN {X 0,Y 488.806,Z 379.599,A -85,B 0,C 180,E1 -6398.263,E2 -6398.263} C_VEL
LIN {X 0,Y 488.818,Z 379.596,A -85,B 0,C 180,E1 -6401.609,E2 -6401.609} C_VEL
LIN {X 0,Y 488.75,Z 379.605,A -85,B 0,C 180,E1 -6404.997,E2 -6404.997} C_VEL
LIN {X 0,Y 488.738,Z 379.608,A -85,B 0,C 180,E1 -6408.439,E2 -6408.439} C_VEL
LIN {X 0,Y 488.692,Z 379.612,A -85,B 0,C 180,E1 -6411.067,E2 -6411.067} C_VEL
LIN {X 0,Y 488.689,Z 379.613,A -85,B 0,C 180,E1 -6413.742,E2 -6413.742} C_VEL
LIN {X 0,Y 488.667,Z 379.617,A -85,B 0,C 180,E1 -6416.473,E2 -6416.473} C_VEL
LIN {X 0,Y 488.374,Z 379.656,A -85,B 0,C 180,E1 -6419.289,E2 -6419.289} C_VEL
LIN {X 0,Y 488.245,Z 379.676,A -85,B 0,C 180,E1 -6420.272,E2 -6420.272} C_VEL
LIN {X 0,Y 488.156,Z 382.599,A -85,B 0,C 180,E1 -6423.163,E2 -6423.163} C_VEL
LIN {X 0,Y 488.109,Z 385.949,A -85,B 0,C 180,E1 -6426.265,E2 -6426.265} C_VEL
LIN {X 0,Y 488.071,Z 389.236,A -85,B 0,C 180,E1 -6429.309,E2 -6429.309} C_VEL
LIN {X 0,Y 488.026,Z 392.852,A -85,B 0,C 180,E1 -6432.591,E2 -6432.591} C_VEL
LIN {X 0,Y 487.965,Z 396.726,A -85,B 0,C 180,E1 -6436.059,E2 -6436.059} C_VEL
LIN {X 0,Y 488.005,Z 398.233,A -85,B 0,C 180,E1 -6437.402,E2 -6437.402} C_VEL
LIN {X 0,Y 490.663,Z 410.863,A -85,B 0,C 180,E1 -6437.851,E2 -6437.851} C_VEL
LIN {X 0,Y 490.677,Z 420.023,A -85,B 0,C 180,E1 -6438.22,E2 -6438.22} C_VEL
LIN {X 0,Y 490.311,Z 432.219,A -85,B 0,C 180,E1 -6438.856,E2 -6438.856} C_VEL
LIN {X 0,Y 489.932,Z 443.691,A -85,B 0,C 180,E1 -6439.63,E2 -6439.63} C_VEL
LIN {X 0,Y 489.524,Z 454.545,A -85,B 0,C 180,E1 -6440.56,E2 -6440.56} C_VEL
LIN {X 0,Y 489.164,Z 464.187,A -85,B 0,C 180,E1 -6441.584,E2 -6441.584} C_VEL
LIN {X 0,Y 488.809,Z 472.285,A -85,B 0,C 180,E1 -6442.63,E2 -6442.63} C_VEL
LIN {X 0,Y 488.52,Z 480.048,A -85,B 0,C 180,E1 -6443.856,E2 -6443.856} C_VEL
LIN {X 0,Y 488.327,Z 486.397,A -85,B 0,C 180,E1 -6445.111,E2 -6445.111} C_VEL
LIN {X 0,Y 488.104,Z 492.312,A -85,B 0,C 180,E1 -6446.62,E2 -6446.62} C_VEL
LIN {X 0,Y 488.004,Z 496.723,A -85,B 0,C 180,E1 -6448.169,E2 -6448.169} C_VEL
LIN {X 0,Y 487.884,Z 499.66,A -85,B 0,C 180,E1 -6449.794,E2 -6449.794} C_VEL
LIN {X 0,Y 487.851,Z 500.622,A -85,B 0,C 180,E1 -6450.673,E2 -6450.673} C_VEL
LIN {X 0,Y 487.84,Z 501.103,A -85,B 0,C 180,E1 -6451.615,E2 -6451.615} C_VEL
LIN {X 0,Y 487.851,Z 501.104,A -85,B 0,C 180,E1 -6452.55,E2 -6452.55} C_VEL
LIN {X 0,Y 487.846,Z 500.604,A -85,B 0,C 180,E1 -6453.476,E2 -6453.476} C_VEL
LIN {X 0,Y 487.955,Z 498.426,A -85,B 0,C 180,E1 -6455.135,E2 -6455.135} C_VEL
LIN {X 0,Y 488.086,Z 494.925,A -85,B 0,C 180,E1 -6456.674,E2 -6456.674} C_VEL
LIN {X 0,Y 488.207,Z 490.531,A -85,B 0,C 180,E1 -6458.021,E2 -6458.021} C_VEL
LIN {X 0,Y 488.355,Z 485.186,A -85,B 0,C 180,E1 -6459.284,E2 -6459.284} C_VEL
LIN {X 0,Y 488.626,Z 477.661,A -85,B 0,C 180,E1 -6460.683,E2 -6460.683} C_VEL
LIN {X 0,Y 488.927,Z 469.817,A -85,B 0,C 180,E1 -6461.844,E2 -6461.844} C_VEL
LIN {X 0,Y 489.347,Z 460.244,A -85,B 0,C 180,E1 -6462.986,E2 -6462.986} C_VEL
LIN {X 0,Y 489.733,Z 449.39,A -85,B 0,C 180,E1 -6464.031,E2 -6464.031} C_VEL
LIN {X 0,Y 490.108,Z 438.956,A -85,B 0,C 180,E1 -6464.83,E2 -6464.83} C_VEL
LIN {X 0,Y 490.518,Z 426.347,A -85,B 0,C 180,E1 -6465.586,E2 -6465.586} C_VEL
LIN {X 0,Y 490.894,Z 414.304,A -85,B 0,C 180,E1 -6466.126,E2 -6466.126} C_VEL
LIN {X 0,Y 490.219,Z 407.922,A -85,B 0,C 180,E1 -6466.371,E2 -6466.371} C_VEL
LIN {X 0,Y 488.077,Z 399.023,A -85,B 0,C 180,E1 -6466.707,E2 -6466.707} C_VEL
LIN {X 0,Y 488.125,Z 396.367,A -85,B 0,C 180,E1 -6469.213,E2 -6469.213} C_VEL
LIN {X 0,Y 488.194,Z 392.895,A -85,B 0,C 180,E1 -6472.556,E2 -6472.556} C_VEL
LIN {X 0,Y 488.33,Z 389.515,A -85,B 0,C 180,E1 -6475.874,E2 -6475.874} C_VEL
LIN {X 0,Y 488.457,Z 386.168,A -85,B 0,C 180,E1 -6479.176,E2 -6479.176} C_VEL
LIN {X 0,Y 488.657,Z 384.507,A -85,B 0,C 180,E1 -6480.825,E2 -6480.825} C_VEL
LIN {X 0,Y 488.655,Z 380.419,A -85,B 0,C 180,E1 -6484.951,E2 -6484.951} C_VEL
LIN {X 0,Y 488.623,Z 379.624,A -85,B 0,C 180,E1 -6485.779,E2 -6485.779} C_VEL
LIN {X 0,Y 488.758,Z 379.607,A -85,B 0,C 180,E1 -6488.268,E2 -6488.268} C_VEL
LIN {X 0,Y 488.802,Z 379.601,A -85,B 0,C 180,E1 -6491.613,E2 -6491.613} C_VEL
LIN {X 0,Y 488.729,Z 379.608,A -85,B 0,C 180,E1 -6495.002,E2 -6495.002} C_VEL
LIN {X 0,Y 488.732,Z 379.606,A -85,B 0,C 180,E1 -6498.444,E2 -6498.444} C_VEL
LIN {X 0,Y 488.709,Z 379.61,A -85,B 0,C 180,E1 -6501.071,E2 -6501.071} C_VEL
LIN {X 0,Y 488.683,Z 379.615,A -85,B 0,C 180,E1 -6503.747,E2 -6503.747} C_VEL
LIN {X 0,Y 488.767,Z 379.603,A -85,B 0,C 180,E1 -6506.948,E2 -6506.948} C_VEL
LIN {X 0,Y 488.689,Z 379.612,A -85,B 0,C 180,E1 -6510.368,E2 -6510.368} C_VEL
LIN {X 0,Y 488.707,Z 379.61,A -85,B 0,C 180,E1 -6513.488,E2 -6513.488} C_VEL
LIN {X 0,Y 488.666,Z 379.615,A -85,B 0,C 180,E1 -6516.359,E2 -6516.359} C_VEL
LIN {X 0,Y 488.725,Z 379.609,A -85,B 0,C 180,E1 -6519.253,E2 -6519.253} C_VEL
LIN {X 0,Y 488.71,Z 379.611,A -85,B 0,C 180,E1 -6522.524,E2 -6522.524} C_VEL
LIN {X 0,Y 488.69,Z 379.613,A -85,B 0,C 180,E1 -6525.202,E2 -6525.202} C_VEL
LIN {X 0,Y 488.713,Z 379.613,A -85,B 0,C 180,E1 -6527.483,E2 -6527.483} C_VEL
LIN {X 0,Y 488.732,Z 379.621,A -85,B 0,C 180,E1 -6529.682,E2 -6529.682} C_VEL
LIN {X 0,Y 489.55,Z 384.445,A -85,B 0,C 180,E1 -6532.147,E2 -6532.147} C_VEL
LIN {X 0,Y 490.171,Z 388.414,A -85,B 0,C 180,E1 -6534,E2 -6534} C_VEL
LIN {X 0,Y 489.928,Z 393.898,A -85,B 0,C 180,E1 -6536.306,E2 -6536.306} C_VEL
LIN {X 0,Y 489.442,Z 402.024,A -85,B 0,C 180,E1 -6539.492,E2 -6539.492} C_VEL
LIN {X 0,Y 489.014,Z 411.626,A -85,B 0,C 180,E1 -6543.006,E2 -6543.006} C_VEL
LIN {X 0,Y 488.77,Z 419.669,A -85,B 0,C 180,E1 -6545.812,E2 -6545.812} C_VEL
LIN {X 0,Y 488.59,Z 427.626,A -85,B 0,C 180,E1 -6548.486,E2 -6548.486} C_VEL
LIN {X 0,Y 488.43,Z 435.625,A -85,B 0,C 180,E1 -6551.114,E2 -6551.114} C_VEL
LIN {X 0,Y 488.291,Z 445.027,A -85,B 0,C 180,E1 -6554.133,E2 -6554.133} C_VEL
LIN {X 0,Y 488.222,Z 448.648,A -85,B 0,C 180,E1 -6555.28,E2 -6555.28} C_VEL
LIN {X 0,Y 490.078,Z 462.676,A -85,B 0,C 180,E1 -6555.695,E2 -6555.695} C_VEL
LIN {X 0,Y 490.671,Z 466.871,A -85,B 0,C 180,E1 -6555.858,E2 -6555.858} C_VEL
LIN {X 0,Y 490.309,Z 479.105,A -85,B 0,C 180,E1 -6556.376,E2 -6556.376} C_VEL
LIN {X 0,Y 489.861,Z 491.431,A -85,B 0,C 180,E1 -6557.081,E2 -6557.081} C_VEL
LIN {X 0,Y 489.419,Z 502.421,A -85,B 0,C 180,E1 -6557.881,E2 -6557.881} C_VEL
LIN {X 0,Y 489.102,Z 512.783,A -85,B 0,C 180,E1 -6558.818,E2 -6558.818} C_VEL
LIN {X 0,Y 488.731,Z 522.107,A -85,B 0,C 180,E1 -6559.857,E2 -6559.857} C_VEL
LIN {X 0,Y 488.422,Z 531.193,A -85,B 0,C 180,E1 -6561.105,E2 -6561.105} C_VEL
LIN {X 0,Y 488.215,Z 538.519,A -85,B 0,C 180,E1 -6562.351,E2 -6562.351} C_VEL
LIN {X 0,Y 488.076,Z 543.947,A -85,B 0,C 180,E1 -6563.497,E2 -6563.497} C_VEL
LIN {X 0,Y 488.051,Z 548.277,A -85,B 0,C 180,E1 -6564.632,E2 -6564.632} C_VEL
LIN {X 0,Y 487.953,Z 551.953,A -85,B 0,C 180,E1 -6565.873,E2 -6565.873} C_VEL
LIN {X 0,Y 487.968,Z 553.856,A -85,B 0,C 180,E1 -6566.7,E2 -6566.7} C_VEL
LIN {X 0,Y 487.959,Z 555.28,A -85,B 0,C 180,E1 -6567.527,E2 -6567.527} C_VEL
LIN {X 0,Y 487.834,Z 556.921,A -85,B 0,C 180,E1 -6569.178,E2 -6569.178} C_VEL
LIN {X 0,Y 487.82,Z 557.149,A -85,B 0,C 180,E1 -6570.003,E2 -6570.003} C_VEL
LIN {X 0,Y 487.894,Z 556.333,A -85,B 0,C 180,E1 -6571.654,E2 -6571.654} C_VEL
LIN {X 0,Y 487.96,Z 555.338,A -85,B 0,C 180,E1 -6572.479,E2 -6572.479} C_VEL
LIN {X 0,Y 487.969,Z 553.929,A -85,B 0,C 180,E1 -6573.306,E2 -6573.306} C_VEL
LIN {X 0,Y 487.93,Z 550.964,A -85,B 0,C 180,E1 -6574.547,E2 -6574.547} C_VEL
LIN {X 0,Y 488.053,Z 546.955,A -85,B 0,C 180,E1 -6575.788,E2 -6575.788} C_VEL
LIN {X 0,Y 488.186,Z 540.773,A -85,B 0,C 180,E1 -6577.239,E2 -6577.239} C_VEL
LIN {X 0,Y 488.367,Z 534.028,A -85,B 0,C 180,E1 -6578.485,E2 -6578.485} C_VEL
LIN {X 0,Y 488.614,Z 525.662,A -85,B 0,C 180,E1 -6579.733,E2 -6579.733} C_VEL
LIN {X 0,Y 488.975,Z 517.072,A -85,B 0,C 180,E1 -6580.772,E2 -6580.772} C_VEL
LIN {X 0,Y 489.411,Z 506.484,A -85,B 0,C 180,E1 -6581.811,E2 -6581.811} C_VEL
LIN {X 0,Y 489.686,Z 496.3,A -85,B 0,C 180,E1 -6582.624,E2 -6582.624} C_VEL
LIN {X 0,Y 490.124,Z 484.537,A -85,B 0,C 180,E1 -6583.372,E2 -6583.372} C_VEL
LIN {X 0,Y 490.583,Z 471.428,A -85,B 0,C 180,E1 -6583.992,E2 -6583.992} C_VEL
LIN {X 0,Y 490.49,Z 465.112,A -85,B 0,C 180,E1 -6584.233,E2 -6584.233} C_VEL
LIN {X 0,Y 488.53,Z 451.727,A -85,B 0,C 180,E1 -6584.66,E2 -6584.66} C_VEL
LIN {X 0,Y 488.231,Z 449.314,A -85,B 0,C 180,E1 -6584.726,E2 -6584.726} C_VEL
LIN {X 0,Y 488.397,Z 440.471,A -85,B 0,C 180,E1 -6587.592,E2 -6587.592} C_VEL
LIN {X 0,Y 488.6,Z 430.821,A -85,B 0,C 180,E1 -6590.778,E2 -6590.778} C_VEL
LIN {X 0,Y 488.841,Z 422.053,A -85,B 0,C 180,E1 -6593.74,E2 -6593.74} C_VEL
LIN {X 0,Y 489.082,Z 414.218,A -85,B 0,C 180,E1 -6596.455,E2 -6596.455} C_VEL
LIN {X 0,Y 489.461,Z 405.121,A -85,B 0,C 180,E1 -6599.697,E2 -6599.697} C_VEL
LIN {X 0,Y 489.813,Z 397.365,A -85,B 0,C 180,E1 -6602.554,E2 -6602.554} C_VEL
LIN {X 0,Y 490.168,Z 390.947,A -85,B 0,C 180,E1 -6604.998,E2 -6604.998} C_VEL
LIN {X 0,Y 490.028,Z 387.027,A -85,B 0,C 180,E1 -6606.567,E2 -6606.567} C_VEL
LIN {X 0,Y 488.733,Z 379.609,A -85,B 0,C 180,E1 -6609.788,E2 -6609.788} C_VEL
LIN {X 0,Y 488.677,Z 379.615,A -85,B 0,C 180,E1 -6612.822,E2 -6612.822} C_VEL
LIN {X 0,Y 488.702,Z 379.613,A -85,B 0,C 180,E1 -6615.978,E2 -6615.978} C_VEL
LIN {X 0,Y 488.693,Z 379.614,A -85,B 0,C 180,E1 -6618.582,E2 -6618.582} C_VEL
LIN {X 0,Y 488.686,Z 379.612,A -85,B 0,C 180,E1 -6621.8,E2 -6621.8} C_VEL
LIN {X 0,Y 488.73,Z 379.609,A -85,B 0,C 180,E1 -6625.054,E2 -6625.054} C_VEL
LIN {X 0,Y 488.713,Z 379.61,A -85,B 0,C 180,E1 -6628.047,E2 -6628.047} C_VEL
LIN {X 0,Y 488.721,Z 379.611,A -85,B 0,C 180,E1 -6630.729,E2 -6630.729} C_VEL
LIN {X 0,Y 488.697,Z 379.612,A -85,B 0,C 180,E1 -6633.524,E2 -6633.524} C_VEL
LIN {X 0,Y 488.685,Z 379.614,A -85,B 0,C 180,E1 -6636.254,E2 -6636.254} C_VEL
LIN {X 0,Y 488.759,Z 379.604,A -85,B 0,C 180,E1 -6639.176,E2 -6639.176} C_VEL
LIN {X 0,Y 488.761,Z 379.603,A -85,B 0,C 180,E1 -6641.632,E2 -6641.632} C_VEL
LIN {X 0,Y 488.766,Z 379.604,A -85,B 0,C 180,E1 -6644.999,E2 -6644.999} C_VEL
LIN {X 0,Y 488.815,Z 379.598,A -85,B 0,C 180,E1 -6648.387,E2 -6648.387} C_VEL
LIN {X 0,Y 488.794,Z 379.6,A -85,B 0,C 180,E1 -6651.733,E2 -6651.733} C_VEL
LIN {X 0,Y 488.847,Z 379.592,A -85,B 0,C 180,E1 -6654.223,E2 -6654.223} C_VEL
LIN {X 0,Y 488.966,Z 379.579,A -85,B 0,C 180,E1 -6657.528,E2 -6657.528} C_VEL
LIN {X 0,Y 488.924,Z 379.584,A -85,B 0,C 180,E1 -6660.823,E2 -6660.823} C_VEL
LIN {X 0,Y 488.959,Z 379.579,A -85,B 0,C 180,E1 -6662.471,E2 -6662.471} C_VEL
LIN {X 0,Y 488.837,Z 379.594,A -85,B 0,C 180,E1 -6665.775,E2 -6665.775} C_VEL
LIN {X 0,Y 488.778,Z 379.603,A -85,B 0,C 180,E1 -6668.266,E2 -6668.266} C_VEL
LIN {X 0,Y 488.812,Z 379.596,A -85,B 0,C 180,E1 -6671.611,E2 -6671.611} C_VEL
LIN {X 0,Y 488.766,Z 379.605,A -85,B 0,C 180,E1 -6674.999,E2 -6674.999} C_VEL
LIN {X 0,Y 488.754,Z 379.604,A -85,B 0,C 180,E1 -6678.441,E2 -6678.441} C_VEL
LIN {X 0,Y 488.715,Z 379.61,A -85,B 0,C 180,E1 -6681.069,E2 -6681.069} C_VEL
LIN {X 0,Y 488.682,Z 379.612,A -85,B 0,C 180,E1 -6683.745,E2 -6683.745} C_VEL
LIN {X 0,Y 488.753,Z 379.607,A -85,B 0,C 180,E1 -6686.931,E2 -6686.931} C_VEL
LIN {X 0,Y 488.714,Z 379.609,A -85,B 0,C 180,E1 -6690.361,E2 -6690.361} C_VEL
LIN {X 0,Y 488.74,Z 379.607,A -85,B 0,C 180,E1 -6693.482,E2 -6693.482} C_VEL
LIN {X 0,Y 488.678,Z 379.616,A -85,B 0,C 180,E1 -6696.351,E2 -6696.351} C_VEL
LIN {X 0,Y 488.702,Z 379.611,A -85,B 0,C 180,E1 -6699.253,E2 -6699.253} C_VEL
LIN {X 0,Y 488.702,Z 379.611,A -85,B 0,C 180,E1 -6701.597,E2 -6701.597} C_VEL
LIN {X 0,Y 488.705,Z 379.611,A -85,B 0,C 180,E1 -6704.801,E2 -6704.801} C_VEL
LIN {X 0,Y 488.692,Z 379.612,A -85,B 0,C 180,E1 -6707.472,E2 -6707.472} C_VEL
LIN {X 0,Y 488.704,Z 379.612,A -85,B 0,C 180,E1 -6710.744,E2 -6710.744} C_VEL
LIN {X 0,Y 488.686,Z 379.614,A -85,B 0,C 180,E1 -6713.866,E2 -6713.866} C_VEL
LIN {X 0,Y 488.741,Z 379.606,A -85,B 0,C 180,E1 -6716.875,E2 -6716.875} C_VEL
LIN {X 0,Y 488.725,Z 379.607,A -85,B 0,C 180,E1 -6719.778,E2 -6719.778} C_VEL
LIN {X 0,Y 488.793,Z 379.601,A -85,B 0,C 180,E1 -6723.054,E2 -6723.054} C_VEL
LIN {X 0,Y 488.743,Z 379.607,A -85,B 0,C 180,E1 -6724.326,E2 -6724.326} C_VEL
LIN {X 0,Y 488.098,Z 379.692,A -85,B 0,C 180,E1 -6725.014,E2 -6725.014} C_VEL
LIN {X 0,Y 485.231,Z 380.049,A -85,B 0,C 180,E1 -6726.13,E2 -6726.13} C_VEL
LIN {X 0,Y 482.785,Z 380.35,A -85,B 0,C 180,E1 -6727.03,E2 -6727.03} C_VEL
LIN {X 0,Y 481.726,Z 380.48,A -85,B 0,C 180,E1 -6727.725,E2 -6727.725} C_VEL
LIN {X 0,Y 481.637,Z 380.49,A -85,B 0,C 180,E1 -6727.961,E2 -6727.961} C_VEL
LIN {X 0,Y 481.704,Z 380.483,A -85,B 0,C 180,E1 -6730.39,E2 -6730.39} C_VEL
LIN {X 0,Y 481.685,Z 380.483,A -85,B 0,C 180,E1 -6733.031,E2 -6733.031} C_VEL
LIN {X 0,Y 481.687,Z 380.485,A -85,B 0,C 180,E1 -6735.636,E2 -6735.636} C_VEL
LIN {X 0,Y 481.748,Z 380.479,A -85,B 0,C 180,E1 -6738.212,E2 -6738.212} C_VEL
LIN {X 0,Y 481.758,Z 380.475,A -85,B 0,C 180,E1 -6741.609,E2 -6741.609} C_VEL
LIN {X 0,Y 481.804,Z 380.471,A -85,B 0,C 180,E1 -6744.137,E2 -6744.137} C_VEL
LIN {X 0,Y 481.922,Z 380.457,A -85,B 0,C 180,E1 -6747.49,E2 -6747.49} C_VEL
LIN {X 0,Y 481.898,Z 380.458,A -85,B 0,C 180,E1 -6750.833,E2 -6750.833} C_VEL
LIN {X 0,Y 481.921,Z 380.458,A -85,B 0,C 180,E1 -6752.504,E2 -6752.504} C_VEL
LIN {X 0,Y 481.81,Z 380.47,A -85,B 0,C 180,E1 -6755.857,E2 -6755.857} C_VEL
LIN {X 0,Y 481.752,Z 380.477,A -85,B 0,C 180,E1 -6758.385,E2 -6758.385} C_VEL
LIN {X 0,Y 481.783,Z 380.473,A -85,B 0,C 180,E1 -6761.781,E2 -6761.781} C_VEL
LIN {X 0,Y 481.729,Z 380.479,A -85,B 0,C 180,E1 -6765.221,E2 -6765.221} C_VEL
LIN {X 0,Y 481.696,Z 380.485,A -85,B 0,C 180,E1 -6768.718,E2 -6768.718} C_VEL
LIN {X 0,Y 481.634,Z 380.492,A -85,B 0,C 180,E1 -6771.391,E2 -6771.391} C_VEL
LIN {X 0,Y 481.668,Z 380.49,A -85,B 0,C 180,E1 -6774.109,E2 -6774.109} C_VEL
LIN {X 0,Y 481.624,Z 380.493,A -85,B 0,C 180,E1 -6776.891,E2 -6776.891} C_VEL
LIN {X 0,Y 481.274,Z 380.542,A -85,B 0,C 180,E1 -6779.764,E2 -6779.764} C_VEL
LIN {X 0,Y 481.144,Z 380.711,A -85,B 0,C 180,E1 -6780.742,E2 -6780.742} C_VEL
LIN {X 0,Y 481.084,Z 383.849,A -85,B 0,C 180,E1 -6783.715,E2 -6783.715} C_VEL
LIN {X 0,Y 481.016,Z 387.157,A -85,B 0,C 180,E1 -6786.796,E2 -6786.796} C_VEL
LIN {X 0,Y 481,Z 390.636,A -85,B 0,C 180,E1 -6790.002,E2 -6790.002} C_VEL
LIN {X 0,Y 480.906,Z 394.325,A -85,B 0,C 180,E1 -6793.376,E2 -6793.376} C_VEL
LIN {X 0,Y 480.894,Z 397.928,A -85,B 0,C 180,E1 -6796.618,E2 -6796.618} C_VEL
LIN {X 0,Y 480.915,Z 398.625,A -85,B 0,C 180,E1 -6797.188,E2 -6797.188} C_VEL
LIN {X 0,Y 483.752,Z 411.624,A -85,B 0,C 180,E1 -6797.663,E2 -6797.663} C_VEL
LIN {X 0,Y 483.831,Z 419.839,A -85,B 0,C 180,E1 -6797.999,E2 -6797.999} C_VEL
LIN {X 0,Y 483.413,Z 432.376,A -85,B 0,C 180,E1 -6798.657,E2 -6798.657} C_VEL
LIN {X 0,Y 483.028,Z 443.005,A -85,B 0,C 180,E1 -6799.376,E2 -6799.376} C_VEL
LIN {X 0,Y 482.606,Z 453.714,A -85,B 0,C 180,E1 -6800.28,E2 -6800.28} C_VEL
LIN {X 0,Y 482.245,Z 462.553,A -85,B 0,C 180,E1 -6801.197,E2 -6801.197} C_VEL
LIN {X 0,Y 481.915,Z 470.782,A -85,B 0,C 180,E1 -6802.23,E2 -6802.23} C_VEL
LIN {X 0,Y 481.603,Z 478.282,A -85,B 0,C 180,E1 -6803.373,E2 -6803.373} C_VEL
LIN {X 0,Y 481.329,Z 484.833,A -85,B 0,C 180,E1 -6804.595,E2 -6804.595} C_VEL
LIN {X 0,Y 481.156,Z 489.967,A -85,B 0,C 180,E1 -6805.783,E2 -6805.783} C_VEL
LIN {X 0,Y 480.993,Z 494.962,A -85,B 0,C 180,E1 -6807.275,E2 -6807.275} C_VEL
LIN {X 0,Y 480.915,Z 497.426,A -85,B 0,C 180,E1 -6808.259,E2 -6808.259} C_VEL
LIN {X 0,Y 480.805,Z 499.813,A -85,B 0,C 180,E1 -6809.579,E2 -6809.579} C_VEL
LIN {X 0,Y 480.77,Z 501.411,A -85,B 0,C 180,E1 -6811.284,E2 -6811.284} C_VEL
LIN {X 0,Y 480.747,Z 501.59,A -85,B 0,C 180,E1 -6812.109,E2 -6812.109} C_VEL
LIN {X 0,Y 480.762,Z 501.285,A -85,B 0,C 180,E1 -6813.081,E2 -6813.081} C_VEL
LIN {X 0,Y 480.79,Z 500.555,A -85,B 0,C 180,E1 -6813.991,E2 -6813.991} C_VEL
LIN {X 0,Y 480.855,Z 499.196,A -85,B 0,C 180,E1 -6814.97,E2 -6814.97} C_VEL
LIN {X 0,Y 480.99,Z 496.44,A -85,B 0,C 180,E1 -6816.309,E2 -6816.309} C_VEL
LIN {X 0,Y 481.108,Z 492.447,A -85,B 0,C 180,E1 -6817.679,E2 -6817.679} C_VEL
LIN {X 0,Y 481.29,Z 486.748,A -85,B 0,C 180,E1 -6819.143,E2 -6819.143} C_VEL
LIN {X 0,Y 481.51,Z 480.518,A -85,B 0,C 180,E1 -6820.386,E2 -6820.386} C_VEL
LIN {X 0,Y 481.819,Z 473.196,A -85,B 0,C 180,E1 -6821.566,E2 -6821.566} C_VEL
LIN {X 0,Y 482.14,Z 465.299,A -85,B 0,C 180,E1 -6822.614,E2 -6822.614} C_VEL
LIN {X 0,Y 482.608,Z 454.852,A -85,B 0,C 180,E1 -6823.743,E2 -6823.743} C_VEL
LIN {X 0,Y 483.051,Z 443.53,A -85,B 0,C 180,E1 -6824.711,E2 -6824.711} C_VEL
LIN {X 0,Y 483.476,Z 432.156,A -85,B 0,C 180,E1 -6825.479,E2 -6825.479} C_VEL
LIN {X 0,Y 483.844,Z 420.679,A -85,B 0,C 180,E1 -6826.08,E2 -6826.08} C_VEL
LIN {X 0,Y 483.874,Z 412.137,A -85,B 0,C 180,E1 -6826.429,E2 -6826.429} C_VEL
LIN {X 0,Y 481.327,Z 401.04,A -85,B 0,C 180,E1 -6826.853,E2 -6826.853} C_VEL
LIN {X 0,Y 481.027,Z 399.498,A -85,B 0,C 180,E1 -6826.912,E2 -6826.912} C_VEL
LIN {X 0,Y 481.085,Z 397.247,A -85,B 0,C 180,E1 -6829.053,E2 -6829.053} C_VEL
LIN {X 0,Y 481.153,Z 393.747,A -85,B 0,C 180,E1 -6832.447,E2 -6832.447} C_VEL
LIN {X 0,Y 481.286,Z 390.353,A -85,B 0,C 180,E1 -6835.814,E2 -6835.814} C_VEL
LIN {X 0,Y 481.409,Z 387.002,A -85,B 0,C 180,E1 -6839.164,E2 -6839.164} C_VEL
LIN {X 0,Y 481.62,Z 385.318,A -85,B 0,C 180,E1 -6840.837,E2 -6840.837} C_VEL
LIN {X 0,Y 481.625,Z 381.242,A -85,B 0,C 180,E1 -6845.024,E2 -6845.024} C_VEL
LIN {X 0,Y 481.595,Z 380.499,A -85,B 0,C 180,E1 -6845.864,E2 -6845.864} C_VEL
LIN {X 0,Y 481.731,Z 380.484,A -85,B 0,C 180,E1 -6847.546,E2 -6847.546} C_VEL
LIN {X 0,Y 481.697,Z 380.486,A -85,B 0,C 180,E1 -6850.084,E2 -6850.084} C_VEL
LIN {X 0,Y 481.712,Z 380.482,A -85,B 0,C 180,E1 -6852.642,E2 -6852.642} C_VEL
LIN {X 0,Y 481.683,Z 380.487,A -85,B 0,C 180,E1 -6856.095,E2 -6856.095} C_VEL
LIN {X 0,Y 481.683,Z 380.485,A -85,B 0,C 180,E1 -6858.724,E2 -6858.724} C_VEL
LIN {X 0,Y 481.644,Z 380.489,A -85,B 0,C 180,E1 -6861.395,E2 -6861.395} C_VEL
LIN {X 0,Y 481.661,Z 380.487,A -85,B 0,C 180,E1 -6864.115,E2 -6864.115} C_VEL
LIN {X 0,Y 481.72,Z 380.48,A -85,B 0,C 180,E1 -6867.143,E2 -6867.143} C_VEL
LIN {X 0,Y 481.658,Z 380.49,A -85,B 0,C 180,E1 -6869.743,E2 -6869.743} C_VEL
LIN {X 0,Y 481.644,Z 380.491,A -85,B 0,C 180,E1 -6872.677,E2 -6872.677} C_VEL
LIN {X 0,Y 481.618,Z 380.495,A -85,B 0,C 180,E1 -6875.712,E2 -6875.712} C_VEL
LIN {X 0,Y 481.697,Z 380.484,A -85,B 0,C 180,E1 -6879.358,E2 -6879.358} C_VEL
LIN {X 0,Y 481.652,Z 380.49,A -85,B 0,C 180,E1 -6882.161,E2 -6882.161} C_VEL
LIN {X 0,Y 481.638,Z 380.493,A -85,B 0,C 180,E1 -6884.461,E2 -6884.461} C_VEL
LIN {X 0,Y 481.668,Z 380.489,A -85,B 0,C 180,E1 -6886.849,E2 -6886.849} C_VEL
LIN {X 0,Y 481.696,Z 380.546,A -85,B 0,C 180,E1 -6889.349,E2 -6889.349} C_VEL
LIN {X 0,Y 482.679,Z 386.222,A -85,B 0,C 180,E1 -6892.305,E2 -6892.305} C_VEL
LIN {X 0,Y 483.207,Z 389.637,A -85,B 0,C 180,E1 -6893.915,E2 -6893.915} C_VEL
LIN {X 0,Y 482.936,Z 395.513,A -85,B 0,C 180,E1 -6896.432,E2 -6896.432} C_VEL
LIN {X 0,Y 482.363,Z 404.024,A -85,B 0,C 180,E1 -6899.828,E2 -6899.828} C_VEL
LIN {X 0,Y 481.945,Z 412.895,A -85,B 0,C 180,E1 -6903.128,E2 -6903.128} C_VEL
LIN {X 0,Y 481.717,Z 420.703,A -85,B 0,C 180,E1 -6905.893,E2 -6905.893} C_VEL
LIN {X 0,Y 481.503,Z 430.045,A -85,B 0,C 180,E1 -6909.091,E2 -6909.091} C_VEL
LIN {X 0,Y 481.268,Z 439.24,A -85,B 0,C 180,E1 -6912.145,E2 -6912.145} C_VEL
LIN {X 0,Y 481.139,Z 448.207,A -85,B 0,C 180,E1 -6915.058,E2 -6915.058} C_VEL
LIN {X 0,Y 483.023,Z 462.602,A -85,B 0,C 180,E1 -6915.495,E2 -6915.495} C_VEL
LIN {X 0,Y 483.684,Z 469.16,A -85,B 0,C 180,E1 -6915.757,E2 -6915.757} C_VEL
LIN {X 0,Y 483.261,Z 481.58,A -85,B 0,C 180,E1 -6916.334,E2 -6916.334} C_VEL
LIN {X 0,Y 482.773,Z 494.189,A -85,B 0,C 180,E1 -6917.112,E2 -6917.112} C_VEL
LIN {X 0,Y 482.308,Z 504.785,A -85,B 0,C 180,E1 -6917.947,E2 -6917.947} C_VEL
LIN {X 0,Y 481.991,Z 514.265,A -85,B 0,C 180,E1 -6918.864,E2 -6918.864} C_VEL
LIN {X 0,Y 481.597,Z 523.266,A -85,B 0,C 180,E1 -6919.918,E2 -6919.918} C_VEL
LIN {X 0,Y 481.301,Z 532.074,A -85,B 0,C 180,E1 -6921.184,E2 -6921.184} C_VEL
LIN {X 0,Y 481.103,Z 539.106,A -85,B 0,C 180,E1 -6922.449,E2 -6922.449} C_VEL
LIN {X 0,Y 480.936,Z 545.145,A -85,B 0,C 180,E1 -6923.813,E2 -6923.813} C_VEL
LIN {X 0,Y 480.904,Z 549.179,A -85,B 0,C 180,E1 -6924.973,E2 -6924.973} C_VEL
LIN {X 0,Y 480.852,Z 551.525,A -85,B 0,C 180,E1 -6925.812,E2 -6925.812} C_VEL
LIN {X 0,Y 480.893,Z 553.435,A -85,B 0,C 180,E1 -6926.652,E2 -6926.652} C_VEL
LIN {X 0,Y 480.869,Z 554.863,A -85,B 0,C 180,E1 -6927.49,E2 -6927.49} C_VEL
LIN {X 0,Y 480.825,Z 555.886,A -85,B 0,C 180,E1 -6928.328,E2 -6928.328} C_VEL
LIN {X 0,Y 480.76,Z 556.514,A -85,B 0,C 180,E1 -6929.165,E2 -6929.165} C_VEL
LIN {X 0,Y 480.744,Z 556.743,A -85,B 0,C 180,E1 -6930.003,E2 -6930.003} C_VEL
LIN {X 0,Y 480.825,Z 555.932,A -85,B 0,C 180,E1 -6931.678,E2 -6931.678} C_VEL
LIN {X 0,Y 480.87,Z 554.935,A -85,B 0,C 180,E1 -6932.516,E2 -6932.516} C_VEL
LIN {X 0,Y 480.894,Z 553.527,A -85,B 0,C 180,E1 -6933.354,E2 -6933.354} C_VEL
LIN {X 0,Y 480.848,Z 550.56,A -85,B 0,C 180,E1 -6934.614,E2 -6934.614} C_VEL
LIN {X 0,Y 480.954,Z 546.546,A -85,B 0,C 180,E1 -6935.874,E2 -6935.874} C_VEL
LIN {X 0,Y 481.112,Z 540.359,A -85,B 0,C 180,E1 -6937.346,E2 -6937.346} C_VEL
LIN {X 0,Y 481.309,Z 533.608,A -85,B 0,C 180,E1 -6938.611,E2 -6938.611} C_VEL
LIN {X 0,Y 481.568,Z 525.235,A -85,B 0,C 180,E1 -6939.877,E2 -6939.877} C_VEL
LIN {X 0,Y 481.951,Z 516.634,A -85,B 0,C 180,E1 -6940.931,E2 -6940.931} C_VEL
LIN {X 0,Y 482.398,Z 506.224,A -85,B 0,C 180,E1 -6941.968,E2 -6941.968} C_VEL
LIN {X 0,Y 482.731,Z 495.85,A -85,B 0,C 180,E1 -6942.809,E2 -6942.809} C_VEL
LIN {X 0,Y 483.185,Z 484.072,A -85,B 0,C 180,E1 -6943.567,E2 -6943.567} C_VEL
LIN {X 0,Y 483.69,Z 470.962,A -85,B 0,C 180,E1 -6944.196,E2 -6944.196} C_VEL
LIN {X 0,Y 483.372,Z 464.629,A -85,B 0,C 180,E1 -6944.447,E2 -6944.447} C_VEL
LIN {X 0,Y 481.488,Z 451.376,A -85,B 0,C 180,E1 -6944.877,E2 -6944.877} C_VEL
LIN {X 0,Y 481.162,Z 448.972,A -85,B 0,C 180,E1 -6944.948,E2 -6944.948} C_VEL
LIN {X 0,Y 481.323,Z 440.166,A -85,B 0,C 180,E1 -6947.859,E2 -6947.859} C_VEL
LIN {X 0,Y 481.54,Z 431.064,A -85,B 0,C 180,E1 -6950.921,E2 -6950.921} C_VEL
LIN {X 0,Y 481.85,Z 421.82,A -85,B 0,C 180,E1 -6954.106,E2 -6954.106} C_VEL
LIN {X 0,Y 482.09,Z 413.987,A -85,B 0,C 180,E1 -6956.87,E2 -6956.87} C_VEL
LIN {X 0,Y 482.455,Z 406.23,A -85,B 0,C 180,E1 -6959.691,E2 -6959.691} C_VEL
LIN {X 0,Y 482.934,Z 397.2,A -85,B 0,C 180,E1 -6963.077,E2 -6963.077} C_VEL
LIN {X 0,Y 483.221,Z 390.807,A -85,B 0,C 180,E1 -6965.577,E2 -6965.577} C_VEL
LIN {X 0,Y 482.782,Z 386.818,A -85,B 0,C 180,E1 -6967.226,E2 -6967.226} C_VEL
LIN {X 0,Y 481.688,Z 380.487,A -85,B 0,C 180,E1 -6970.071,E2 -6970.071} C_VEL
LIN {X 0,Y 481.635,Z 380.492,A -85,B 0,C 180,E1 -6973.303,E2 -6973.303} C_VEL
LIN {X 0,Y 481.665,Z 380.487,A -85,B 0,C 180,E1 -6975.643,E2 -6975.643} C_VEL
LIN {X 0,Y 481.646,Z 380.491,A -85,B 0,C 180,E1 -6978.957,E2 -6978.957} C_VEL
LIN {X 0,Y 481.66,Z 380.487,A -85,B 0,C 180,E1 -6981.995,E2 -6981.995} C_VEL
LIN {X 0,Y 481.694,Z 380.486,A -85,B 0,C 180,E1 -6985.318,E2 -6985.318} C_VEL
LIN {X 0,Y 481.655,Z 380.489,A -85,B 0,C 180,E1 -6988.312,E2 -6988.312} C_VEL
LIN {X 0,Y 481.686,Z 380.485,A -85,B 0,C 180,E1 -6991.217,E2 -6991.217} C_VEL
LIN {X 0,Y 481.658,Z 380.486,A -85,B 0,C 180,E1 -6994.04,E2 -6994.04} C_VEL
LIN {X 0,Y 481.687,Z 380.485,A -85,B 0,C 180,E1 -6996.812,E2 -6996.812} C_VEL
LIN {X 0,Y 481.707,Z 380.482,A -85,B 0,C 180,E1 -6999.503,E2 -6999.503} C_VEL
LIN {X 0,Y 481.703,Z 380.481,A -85,B 0,C 180,E1 -7002.158,E2 -7002.158} C_VEL
LIN {X 0,Y 481.75,Z 380.477,A -85,B 0,C 180,E1 -7004.775,E2 -7004.775} C_VEL
LIN {X 0,Y 481.761,Z 380.476,A -85,B 0,C 180,E1 -7008.215,E2 -7008.215} C_VEL
LIN {X 0,Y 481.749,Z 380.477,A -85,B 0,C 180,E1 -7011.611,E2 -7011.611} C_VEL
LIN {X 0,Y 481.808,Z 380.468,A -85,B 0,C 180,E1 -7014.139,E2 -7014.139} C_VEL
LIN {X 0,Y 481.934,Z 380.455,A -85,B 0,C 180,E1 -7017.492,E2 -7017.492} C_VEL
LIN {X 0,Y 481.948,Z 380.452,A -85,B 0,C 180,E1 -7019.999,E2 -7019.999} C_VEL
LIN {X 0,Y 481.925,Z 380.455,A -85,B 0,C 180,E1 -7022.507,E2 -7022.507} C_VEL
LIN {X 0,Y 481.796,Z 380.471,A -85,B 0,C 180,E1 -7025.86,E2 -7025.86} C_VEL
LIN {X 0,Y 481.737,Z 380.481,A -85,B 0,C 180,E1 -7028.388,E2 -7028.388} C_VEL
LIN {X 0,Y 481.759,Z 380.475,A -85,B 0,C 180,E1 -7031.784,E2 -7031.784} C_VEL
LIN {X 0,Y 481.749,Z 380.477,A -85,B 0,C 180,E1 -7035.223,E2 -7035.223} C_VEL
LIN {X 0,Y 481.715,Z 380.483,A -85,B 0,C 180,E1 -7038.721,E2 -7038.721} C_VEL
LIN {X 0,Y 481.653,Z 380.49,A -85,B 0,C 180,E1 -7041.393,E2 -7041.393} C_VEL
LIN {X 0,Y 481.664,Z 380.487,A -85,B 0,C 180,E1 -7044.113,E2 -7044.113} C_VEL
LIN {X 0,Y 481.717,Z 380.481,A -85,B 0,C 180,E1 -7047.129,E2 -7047.129} C_VEL
LIN {X 0,Y 481.679,Z 380.486,A -85,B 0,C 180,E1 -7049.74,E2 -7049.74} C_VEL
LIN {X 0,Y 481.678,Z 380.487,A -85,B 0,C 180,E1 -7052.673,E2 -7052.673} C_VEL
LIN {X 0,Y 481.638,Z 380.489,A -85,B 0,C 180,E1 -7055.708,E2 -7055.708} C_VEL
LIN {X 0,Y 481.673,Z 380.489,A -85,B 0,C 180,E1 -7058.858,E2 -7058.858} C_VEL
LIN {X 0,Y 481.651,Z 380.491,A -85,B 0,C 180,E1 -7061.91,E2 -7061.91} C_VEL
LIN {X 0,Y 481.658,Z 380.491,A -85,B 0,C 180,E1 -7064.456,E2 -7064.456} C_VEL
LIN {X 0,Y 481.647,Z 380.489,A -85,B 0,C 180,E1 -7067.837,E2 -7067.837} C_VEL
LIN {X 0,Y 481.663,Z 380.488,A -85,B 0,C 180,E1 -7070.652,E2 -7070.652} C_VEL
LIN {X 0,Y 481.633,Z 380.491,A -85,B 0,C 180,E1 -7073.374,E2 -7073.374} C_VEL
LIN {X 0,Y 481.713,Z 380.483,A -85,B 0,C 180,E1 -7076.328,E2 -7076.328} C_VEL
LIN {X 0,Y 481.652,Z 380.489,A -85,B 0,C 180,E1 -7079.415,E2 -7079.415} C_VEL
LIN {X 0,Y 481.7,Z 380.485,A -85,B 0,C 180,E1 -7082.166,E2 -7082.166} C_VEL
LIN {X 0,Y 481.719,Z 380.48,A -85,B 0,C 180,E1 -7084.967,E2 -7084.967} C_VEL
LIN {X 0,Y 481.637,Z 380.49,A -85,B 0,C 180,E1 -7087.961,E2 -7087.961} C_VEL
LIN {X 0,Y 480.968,Z 380.575,A -85,B 0,C 180,E1 -7088.659,E2 -7088.659} C_VEL
LIN {X 0,Y 478.142,Z 380.927,A -85,B 0,C 180,E1 -7089.793,E2 -7089.793} C_VEL
LIN {X 0,Y 475.758,Z 381.224,A -85,B 0,C 180,E1 -7090.707,E2 -7090.707} C_VEL
LIN {X 0,Y 474.736,Z 381.351,A -85,B 0,C 180,E1 -7091.413,E2 -7091.413} C_VEL
LIN {X 0,Y 474.653,Z 381.36,A -85,B 0,C 180,E1 -7091.652,E2 -7091.652} C_VEL
LIN {X 0,Y 474.698,Z 381.356,A -85,B 0,C 180,E1 -7094.542,E2 -7094.542} C_VEL
LIN {X 0,Y 474.702,Z 381.358,A -85,B 0,C 180,E1 -7098.035,E2 -7098.035} C_VEL
LIN {X 0,Y 474.723,Z 381.35,A -85,B 0,C 180,E1 -7101.484,E2 -7101.484} C_VEL
LIN {X 0,Y 474.767,Z 381.347,A -85,B 0,C 180,E1 -7104.049,E2 -7104.049} C_VEL
LIN {X 0,Y 474.888,Z 381.332,A -85,B 0,C 180,E1 -7107.452,E2 -7107.452} C_VEL
LIN {X 0,Y 474.904,Z 381.332,A -85,B 0,C 180,E1 -7109.997,E2 -7109.997} C_VEL
LIN {X 0,Y 474.886,Z 381.334,A -85,B 0,C 180,E1 -7112.541,E2 -7112.541} C_VEL
LIN {X 0,Y 474.772,Z 381.347,A -85,B 0,C 180,E1 -7115.944,E2 -7115.944} C_VEL
LIN {X 0,Y 474.717,Z 381.353,A -85,B 0,C 180,E1 -7118.51,E2 -7118.51} C_VEL
LIN {X 0,Y 474.727,Z 381.354,A -85,B 0,C 180,E1 -7121.958,E2 -7121.958} C_VEL
LIN {X 0,Y 474.686,Z 381.357,A -85,B 0,C 180,E1 -7125.774,E2 -7125.774} C_VEL
LIN {X 0,Y 474.649,Z 381.361,A -85,B 0,C 180,E1 -7129.007,E2 -7129.007} C_VEL
LIN {X 0,Y 474.578,Z 381.372,A -85,B 0,C 180,E1 -7131.725,E2 -7131.725} C_VEL
LIN {X 0,Y 474.646,Z 381.361,A -85,B 0,C 180,E1 -7134.489,E2 -7134.489} C_VEL
LIN {X 0,Y 474.516,Z 381.379,A -85,B 0,C 180,E1 -7137.327,E2 -7137.327} C_VEL
LIN {X 0,Y 474.144,Z 381.432,A -85,B 0,C 180,E1 -7140.258,E2 -7140.258} C_VEL
LIN {X 0,Y 474.086,Z 381.44,A -85,B 0,C 180,E1 -7140.707,E2 -7140.707} C_VEL
LIN {X 0,Y 474,Z 384.692,A -85,B 0,C 180,E1 -7143.871,E2 -7143.871} C_VEL
LIN {X 0,Y 473.967,Z 387.805,A -85,B 0,C 180,E1 -7146.803,E2 -7146.803} C_VEL
LIN {X 0,Y 473.93,Z 390.833,A -85,B 0,C 180,E1 -7149.612,E2 -7149.612} C_VEL
LIN {X 0,Y 473.841,Z 394.548,A -85,B 0,C 180,E1 -7153.015,E2 -7153.015} C_VEL
LIN {X 0,Y 473.838,Z 397.619,A -85,B 0,C 180,E1 -7155.806,E2 -7155.806} C_VEL
LIN {X 0,Y 473.843,Z 398.91,A -85,B 0,C 180,E1 -7156.948,E2 -7156.948} C_VEL
LIN {X 0,Y 477.007,Z 413.535,A -85,B 0,C 180,E1 -7157.52,E2 -7157.52} C_VEL
LIN {X 0,Y 476.767,Z 426.395,A -85,B 0,C 180,E1 -7158.108,E2 -7158.108} C_VEL
LIN {X 0,Y 476.38,Z 437.721,A -85,B 0,C 180,E1 -7158.792,E2 -7158.792} C_VEL
LIN {X 0,Y 475.846,Z 449.556,A -85,B 0,C 180,E1 -7159.701,E2 -7159.701} C_VEL
LIN {X 0,Y 475.441,Z 459.543,A -85,B 0,C 180,E1 -7160.672,E2 -7160.672} C_VEL
LIN {X 0,Y 474.999,Z 469.528,A -85,B 0,C 180,E1 -7161.871,E2 -7161.871} C_VEL
LIN {X 0,Y 474.603,Z 477.723,A -85,B 0,C 180,E1 -7163.088,E2 -7163.088} C_VEL
LIN {X 0,Y 474.296,Z 484.809,A -85,B 0,C 180,E1 -7164.404,E2 -7164.404} C_VEL
LIN {X 0,Y 474.107,Z 490.438,A -85,B 0,C 180,E1 -7165.717,E2 -7165.717} C_VEL
LIN {X 0,Y 473.916,Z 495.42,A -85,B 0,C 180,E1 -7167.231,E2 -7167.231} C_VEL
LIN {X 0,Y 473.77,Z 498.887,A -85,B 0,C 180,E1 -7168.723,E2 -7168.723} C_VEL
LIN {X 0,Y 473.721,Z 500.432,A -85,B 0,C 180,E1 -7169.709,E2 -7169.709} C_VEL
LIN {X 0,Y 473.703,Z 501.699,A -85,B 0,C 180,E1 -7171.076,E2 -7171.076} C_VEL
LIN {X 0,Y 473.688,Z 501.806,A -85,B 0,C 180,E1 -7172.889,E2 -7172.889} C_VEL
LIN {X 0,Y 473.74,Z 500.347,A -85,B 0,C 180,E1 -7174.52,E2 -7174.52} C_VEL
LIN {X 0,Y 473.898,Z 497.877,A -85,B 0,C 180,E1 -7175.932,E2 -7175.932} C_VEL
LIN {X 0,Y 474.024,Z 494.274,A -85,B 0,C 180,E1 -7177.327,E2 -7177.327} C_VEL
LIN {X 0,Y 474.151,Z 489.575,A -85,B 0,C 180,E1 -7178.674,E2 -7178.674} C_VEL
LIN {X 0,Y 474.433,Z 483.183,A -85,B 0,C 180,E1 -7180.081,E2 -7180.081} C_VEL
LIN {X 0,Y 474.715,Z 476.033,A -85,B 0,C 180,E1 -7181.337,E2 -7181.337} C_VEL
LIN {X 0,Y 475.133,Z 467.333,A -85,B 0,C 180,E1 -7182.571,E2 -7182.571} C_VEL
LIN {X 0,Y 475.535,Z 457.477,A -85,B 0,C 180,E1 -7183.693,E2 -7183.693} C_VEL
LIN {X 0,Y 476.049,Z 446.454,A -85,B 0,C 180,E1 -7184.7,E2 -7184.7} C_VEL
LIN {X 0,Y 476.491,Z 435.749,A -85,B 0,C 180,E1 -7185.479,E2 -7185.479} C_VEL
LIN {X 0,Y 476.915,Z 423.975,A -85,B 0,C 180,E1 -7186.146,E2 -7186.146} C_VEL
LIN {X 0,Y 477.021,Z 413.089,A -85,B 0,C 180,E1 -7186.621,E2 -7186.621} C_VEL
LIN {X 0,Y 473.966,Z 399.953,A -85,B 0,C 180,E1 -7187.15,E2 -7187.15} C_VEL
LIN {X 0,Y 473.966,Z 397.269,A -85,B 0,C 180,E1 -7189.751,E2 -7189.751} C_VEL
LIN {X 0,Y 474.092,Z 394.62,A -85,B 0,C 180,E1 -7192.334,E2 -7192.334} C_VEL
LIN {X 0,Y 474.245,Z 391.182,A -85,B 0,C 180,E1 -7195.751,E2 -7195.751} C_VEL
LIN {X 0,Y 474.362,Z 387.833,A -85,B 0,C 180,E1 -7199.152,E2 -7199.152} C_VEL
LIN {X 0,Y 474.584,Z 386.161,A -85,B 0,C 180,E1 -7200.849,E2 -7200.849} C_VEL
LIN {X 0,Y 474.597,Z 382.099,A -85,B 0,C 180,E1 -7205.098,E2 -7205.098} C_VEL
LIN {X 0,Y 474.57,Z 381.375,A -85,B 0,C 180,E1 -7205.951,E2 -7205.951} C_VEL
LIN {X 0,Y 474.684,Z 381.361,A -85,B 0,C 180,E1 -7208.515,E2 -7208.515} C_VEL
LIN {X 0,Y 474.707,Z 381.356,A -85,B 0,C 180,E1 -7211.963,E2 -7211.963} C_VEL
LIN {X 0,Y 474.667,Z 381.359,A -85,B 0,C 180,E1 -7215.779,E2 -7215.779} C_VEL
LIN {X 0,Y 474.634,Z 381.365,A -85,B 0,C 180,E1 -7219.012,E2 -7219.012} C_VEL
LIN {X 0,Y 474.612,Z 381.365,A -85,B 0,C 180,E1 -7221.728,E2 -7221.728} C_VEL
LIN {X 0,Y 474.637,Z 381.361,A -85,B 0,C 180,E1 -7224.495,E2 -7224.495} C_VEL
LIN {X 0,Y 474.667,Z 381.358,A -85,B 0,C 180,E1 -7227.341,E2 -7227.341} C_VEL
LIN {X 0,Y 474.58,Z 381.371,A -85,B 0,C 180,E1 -7230.814,E2 -7230.814} C_VEL
LIN {X 0,Y 474.61,Z 381.367,A -85,B 0,C 180,E1 -7233.987,E2 -7233.987} C_VEL
LIN {X 0,Y 474.553,Z 381.375,A -85,B 0,C 180,E1 -7236.904,E2 -7236.904} C_VEL
LIN {X 0,Y 474.642,Z 381.365,A -85,B 0,C 180,E1 -7239.657,E2 -7239.657} C_VEL
LIN {X 0,Y 474.629,Z 381.368,A -85,B 0,C 180,E1 -7242.933,E2 -7242.933} C_VEL
LIN {X 0,Y 474.597,Z 381.371,A -85,B 0,C 180,E1 -7245.9,E2 -7245.9} C_VEL
LIN {X 0,Y 474.666,Z 381.541,A -85,B 0,C 180,E1 -7249.036,E2 -7249.036} C_VEL
LIN {X 0,Y 475.696,Z 387.443,A -85,B 0,C 180,E1 -7252.189,E2 -7252.189} C_VEL
LIN {X 0,Y 476.205,Z 391.76,A -85,B 0,C 180,E1 -7254.264,E2 -7254.264} C_VEL
LIN {X 0,Y 475.871,Z 397.816,A -85,B 0,C 180,E1 -7256.882,E2 -7256.882} C_VEL
LIN {X 0,Y 475.33,Z 405.117,A -85,B 0,C 180,E1 -7259.825,E2 -7259.825} C_VEL
LIN {X 0,Y 474.909,Z 413.964,A -85,B 0,C 180,E1 -7263.174,E2 -7263.174} C_VEL
LIN {X 0,Y 474.667,Z 421.73,A -85,B 0,C 180,E1 -7265.977,E2 -7265.977} C_VEL
LIN {X 0,Y 474.421,Z 430.891,A -85,B 0,C 180,E1 -7269.178,E2 -7269.178} C_VEL
LIN {X 0,Y 474.177,Z 440.185,A -85,B 0,C 180,E1 -7272.315,E2 -7272.315} C_VEL
LIN {X 0,Y 474.075,Z 447.766,A -85,B 0,C 180,E1 -7274.83,E2 -7274.83} C_VEL
LIN {X 0,Y 475.921,Z 462.126,A -85,B 0,C 180,E1 -7275.273,E2 -7275.273} C_VEL
LIN {X 0,Y 476.807,Z 468.687,A -85,B 0,C 180,E1 -7275.547,E2 -7275.547} C_VEL
LIN {X 0,Y 476.354,Z 481.092,A -85,B 0,C 180,E1 -7276.132,E2 -7276.132} C_VEL
LIN {X 0,Y 475.877,Z 493.121,A -85,B 0,C 180,E1 -7276.879,E2 -7276.879} C_VEL
LIN {X 0,Y 475.355,Z 503.766,A -85,B 0,C 180,E1 -7277.719,E2 -7277.719} C_VEL
LIN {X 0,Y 474.999,Z 513.792,A -85,B 0,C 180,E1 -7278.698,E2 -7278.698} C_VEL
LIN {X 0,Y 474.561,Z 522.797,A -85,B 0,C 180,E1 -7279.767,E2 -7279.767} C_VEL
LIN {X 0,Y 474.25,Z 531.614,A -85,B 0,C 180,E1 -7281.052,E2 -7281.052} C_VEL
LIN {X 0,Y 474.033,Z 538.656,A -85,B 0,C 180,E1 -7282.335,E2 -7282.335} C_VEL
LIN {X 0,Y 473.878,Z 544.048,A -85,B 0,C 180,E1 -7283.55,E2 -7283.55} C_VEL
LIN {X 0,Y 473.838,Z 548.748,A -85,B 0,C 180,E1 -7284.898,E2 -7284.898} C_VEL
LIN {X 0,Y 473.755,Z 551.098,A -85,B 0,C 180,E1 -7285.75,E2 -7285.75} C_VEL
LIN {X 0,Y 473.819,Z 553.014,A -85,B 0,C 180,E1 -7286.602,E2 -7286.602} C_VEL
LIN {X 0,Y 473.783,Z 554.449,A -85,B 0,C 180,E1 -7287.453,E2 -7287.453} C_VEL
LIN {X 0,Y 473.758,Z 555.476,A -85,B 0,C 180,E1 -7288.303,E2 -7288.303} C_VEL
LIN {X 0,Y 473.689,Z 556.107,A -85,B 0,C 180,E1 -7289.153,E2 -7289.153} C_VEL
LIN {X 0,Y 473.67,Z 556.338,A -85,B 0,C 180,E1 -7290.003,E2 -7290.003} C_VEL
LIN {X 0,Y 473.759,Z 555.53,A -85,B 0,C 180,E1 -7291.703,E2 -7291.703} C_VEL
LIN {X 0,Y 473.784,Z 554.533,A -85,B 0,C 180,E1 -7292.554,E2 -7292.554} C_VEL
LIN {X 0,Y 473.82,Z 553.124,A -85,B 0,C 180,E1 -7293.404,E2 -7293.404} C_VEL
LIN {X 0,Y 473.771,Z 550.155,A -85,B 0,C 180,E1 -7294.683,E2 -7294.683} C_VEL
LIN {X 0,Y 473.858,Z 546.137,A -85,B 0,C 180,E1 -7295.962,E2 -7295.962} C_VEL
LIN {X 0,Y 474.021,Z 539.944,A -85,B 0,C 180,E1 -7297.457,E2 -7297.457} C_VEL
LIN {X 0,Y 474.235,Z 533.187,A -85,B 0,C 180,E1 -7298.74,E2 -7298.74} C_VEL
LIN {X 0,Y 474.508,Z 524.806,A -85,B 0,C 180,E1 -7300.025,E2 -7300.025} C_VEL
LIN {X 0,Y 474.92,Z 516.194,A -85,B 0,C 180,E1 -7301.094,E2 -7301.094} C_VEL
LIN {X 0,Y 475.383,Z 506.016,A -85,B 0,C 180,E1 -7302.125,E2 -7302.125} C_VEL
LIN {X 0,Y 475.806,Z 495.095,A -85,B 0,C 180,E1 -7303.021,E2 -7303.021} C_VEL
LIN {X 0,Y 476.268,Z 483.576,A -85,B 0,C 180,E1 -7303.768,E2 -7303.768} C_VEL
LIN {X 0,Y 476.783,Z 470.44,A -85,B 0,C 180,E1 -7304.406,E2 -7304.406} C_VEL
LIN {X 0,Y 476.397,Z 465.195,A -85,B 0,C 180,E1 -7304.623,E2 -7304.623} C_VEL
LIN {X 0,Y 474.518,Z 451.796,A -85,B 0,C 180,E1 -7305.076,E2 -7305.076} C_VEL
LIN {X 0,Y 474.095,Z 448.611,A -85,B 0,C 180,E1 -7305.176,E2 -7305.176} C_VEL
LIN {X 0,Y 474.327,Z 438.739,A -85,B 0,C 180,E1 -7308.508,E2 -7308.508} C_VEL
LIN {X 0,Y 474.54,Z 429.383,A -85,B 0,C 180,E1 -7311.734,E2 -7311.734} C_VEL
LIN {X 0,Y 474.833,Z 421.561,A -85,B 0,C 180,E1 -7314.486,E2 -7314.486} C_VEL
LIN {X 0,Y 475.181,Z 412.424,A -85,B 0,C 180,E1 -7317.792,E2 -7317.792} C_VEL
LIN {X 0,Y 475.593,Z 403.81,A -85,B 0,C 180,E1 -7321.008,E2 -7321.008} C_VEL
LIN {X 0,Y 476.129,Z 395.42,A -85,B 0,C 180,E1 -7324.248,E2 -7324.248} C_VEL
LIN {X 0,Y 476.164,Z 390.625,A -85,B 0,C 180,E1 -7326.187,E2 -7326.187} C_VEL
LIN {X 0,Y 475.136,Z 384.25,A -85,B 0,C 180,E1 -7328.952,E2 -7328.952} C_VEL
LIN {X 0,Y 474.655,Z 381.363,A -85,B 0,C 180,E1 -7330.262,E2 -7330.262} C_VEL
LIN {X 0,Y 474.601,Z 381.368,A -85,B 0,C 180,E1 -7333.48,E2 -7333.48} C_VEL
LIN {X 0,Y 474.601,Z 381.367,A -85,B 0,C 180,E1 -7336.522,E2 -7336.522} C_VEL
LIN {X 0,Y 474.608,Z 381.367,A -85,B 0,C 180,E1 -7339.341,E2 -7339.341} C_VEL
LIN {X 0,Y 474.618,Z 381.365,A -85,B 0,C 180,E1 -7341.706,E2 -7341.706} C_VEL
LIN {X 0,Y 474.631,Z 381.363,A -85,B 0,C 180,E1 -7344.726,E2 -7344.726} C_VEL
LIN {X 0,Y 474.64,Z 381.364,A -85,B 0,C 180,E1 -7347.787,E2 -7347.787} C_VEL
LIN {X 0,Y 474.619,Z 381.367,A -85,B 0,C 180,E1 -7350.889,E2 -7350.889} C_VEL
LIN {X 0,Y 474.605,Z 381.366,A -85,B 0,C 180,E1 -7353.624,E2 -7353.624} C_VEL
LIN {X 0,Y 474.647,Z 381.362,A -85,B 0,C 180,E1 -7356.642,E2 -7356.642} C_VEL
LIN {X 0,Y 474.666,Z 381.36,A -85,B 0,C 180,E1 -7360.089,E2 -7360.089} C_VEL
LIN {X 0,Y 474.649,Z 381.364,A -85,B 0,C 180,E1 -7362.774,E2 -7362.774} C_VEL
LIN {X 0,Y 474.65,Z 381.362,A -85,B 0,C 180,E1 -7365.42,E2 -7365.42} C_VEL
LIN {X 0,Y 474.715,Z 381.353,A -85,B 0,C 180,E1 -7368.037,E2 -7368.037} C_VEL
LIN {X 0,Y 474.721,Z 381.352,A -85,B 0,C 180,E1 -7371.486,E2 -7371.486} C_VEL
LIN {X 0,Y 474.772,Z 381.345,A -85,B 0,C 180,E1 -7374.052,E2 -7374.052} C_VEL
LIN {X 0,Y 474.9,Z 381.331,A -85,B 0,C 180,E1 -7377.455,E2 -7377.455} C_VEL
LIN {X 0,Y 474.918,Z 381.328,A -85,B 0,C 180,E1 -7379.999,E2 -7379.999} C_VEL
LIN {X 0,Y 474.891,Z 381.331,A -85,B 0,C 180,E1 -7382.544,E2 -7382.544} C_VEL
LIN {X 0,Y 474.757,Z 381.348,A -85,B 0,C 180,E1 -7385.947,E2 -7385.947} C_VEL
LIN {X 0,Y 474.712,Z 381.355,A -85,B 0,C 180,E1 -7388.513,E2 -7388.513} C_VEL
LIN {X 0,Y 474.712,Z 381.353,A -85,B 0,C 180,E1 -7391.961,E2 -7391.961} C_VEL
LIN {X 0,Y 474.707,Z 381.353,A -85,B 0,C 180,E1 -7395.455,E2 -7395.455} C_VEL
LIN {X 0,Y 474.67,Z 381.36,A -85,B 0,C 180,E1 -7399.009,E2 -7399.009} C_VEL
LIN {X 0,Y 474.596,Z 381.368,A -85,B 0,C 180,E1 -7401.728,E2 -7401.728} C_VEL
LIN {X 0,Y 474.646,Z 381.364,A -85,B 0,C 180,E1 -7404.493,E2 -7404.493} C_VEL
LIN {X 0,Y 474.681,Z 381.356,A -85,B 0,C 180,E1 -7407.331,E2 -7407.331} C_VEL
LIN {X 0,Y 474.61,Z 381.368,A -85,B 0,C 180,E1 -7410.808,E2 -7410.808} C_VEL
LIN {X 0,Y 474.644,Z 381.363,A -85,B 0,C 180,E1 -7413.982,E2 -7413.982} C_VEL
LIN {X 0,Y 474.571,Z 381.371,A -85,B 0,C 180,E1 -7416.896,E2 -7416.896} C_VEL
LIN {X 0,Y 474.611,Z 381.364,A -85,B 0,C 180,E1 -7419.642,E2 -7419.642} C_VEL
LIN {X 0,Y 474.604,Z 381.368,A -85,B 0,C 180,E1 -7422.231,E2 -7422.231} C_VEL
LIN {X 0,Y 474.62,Z 381.365,A -85,B 0,C 180,E1 -7425.296,E2 -7425.296} C_VEL
LIN {X 0,Y 474.619,Z 381.366,A -85,B 0,C 180,E1 -7428.212,E2 -7428.212} C_VEL
LIN {X 0,Y 474.615,Z 381.365,A -85,B 0,C 180,E1 -7431.541,E2 -7431.541} C_VEL
LIN {X 0,Y 474.632,Z 381.365,A -85,B 0,C 180,E1 -7434.724,E2 -7434.724} C_VEL
LIN {X 0,Y 474.638,Z 381.363,A -85,B 0,C 180,E1 -7437.785,E2 -7437.785} C_VEL
LIN {X 0,Y 474.624,Z 381.364,A -85,B 0,C 180,E1 -7440.883,E2 -7440.883} C_VEL
LIN {X 0,Y 474.662,Z 381.36,A -85,B 0,C 180,E1 -7443.626,E2 -7443.626} C_VEL
LIN {X 0,Y 474.636,Z 381.363,A -85,B 0,C 180,E1 -7446.639,E2 -7446.639} C_VEL
LIN {X 0,Y 474.654,Z 381.363,A -85,B 0,C 180,E1 -7450.087,E2 -7450.087} C_VEL
LIN {X 0,Y 474.653,Z 381.36,A -85,B 0,C 180,E1 -7451.652,E2 -7451.652} C_VEL
LIN {X 0,Y 473.988,Z 381.446,A -85,B 0,C 180,E1 -7452.361,E2 -7452.361} C_VEL
LIN {X 0,Y 471.138,Z 381.801,A -85,B 0,C 180,E1 -7453.512,E2 -7453.512} C_VEL
LIN {X 0,Y 468.724,Z 382.101,A -85,B 0,C 180,E1 -7454.441,E2 -7454.441} C_VEL
LIN {X 0,Y 467.682,Z 382.229,A -85,B 0,C 180,E1 -7455.158,E2 -7455.158} C_VEL
LIN {X 0,Y 467.595,Z 382.239,A -85,B 0,C 180,E1 -7455.401,E2 -7455.401} C_VEL
LIN {X 0,Y 467.65,Z 382.233,A -85,B 0,C 180,E1 -7458.731,E2 -7458.731} C_VEL
LIN {X 0,Y 467.744,Z 382.223,A -85,B 0,C 180,E1 -7462.225,E2 -7462.225} C_VEL
LIN {X 0,Y 467.717,Z 382.224,A -85,B 0,C 180,E1 -7464.824,E2 -7464.824} C_VEL
LIN {X 0,Y 467.853,Z 382.208,A -85,B 0,C 180,E1 -7467.414,E2 -7467.414} C_VEL
LIN {X 0,Y 467.874,Z 382.208,A -85,B 0,C 180,E1 -7469.997,E2 -7469.997} C_VEL
LIN {X 0,Y 467.852,Z 382.21,A -85,B 0,C 180,E1 -7472.58,E2 -7472.58} C_VEL
LIN {X 0,Y 467.736,Z 382.223,A -85,B 0,C 180,E1 -7476.034,E2 -7476.034} C_VEL
LIN {X 0,Y 467.671,Z 382.23,A -85,B 0,C 180,E1 -7478.639,E2 -7478.639} C_VEL
LIN {X 0,Y 467.67,Z 382.233,A -85,B 0,C 180,E1 -7482.141,E2 -7482.141} C_VEL
LIN {X 0,Y 467.651,Z 382.234,A -85,B 0,C 180,E1 -7485.89,E2 -7485.89} C_VEL
LIN {X 0,Y 467.607,Z 382.238,A -85,B 0,C 180,E1 -7489.304,E2 -7489.304} C_VEL
LIN {X 0,Y 467.522,Z 382.25,A -85,B 0,C 180,E1 -7492.07,E2 -7492.07} C_VEL
LIN {X 0,Y 467.58,Z 382.24,A -85,B 0,C 180,E1 -7494.884,E2 -7494.884} C_VEL
LIN {X 0,Y 467.416,Z 382.265,A -85,B 0,C 180,E1 -7497.778,E2 -7497.778} C_VEL
LIN {X 0,Y 467.022,Z 382.32,A -85,B 0,C 180,E1 -7500.935,E2 -7500.935} C_VEL
LIN {X 0,Y 466.915,Z 385.637,A -85,B 0,C 180,E1 -7504.122,E2 -7504.122} C_VEL
LIN {X 0,Y 466.895,Z 388.771,A -85,B 0,C 180,E1 -7507.082,E2 -7507.082} C_VEL
LIN {X 0,Y 466.843,Z 392.251,A -85,B 0,C 180,E1 -7510.335,E2 -7510.335} C_VEL
LIN {X 0,Y 466.765,Z 396.067,A -85,B 0,C 180,E1 -7513.831,E2 -7513.831} C_VEL
LIN {X 0,Y 466.785,Z 399.351,A -85,B 0,C 180,E1 -7516.741,E2 -7516.741} C_VEL
LIN {X 0,Y 469.932,Z 413.186,A -85,B 0,C 180,E1 -7517.278,E2 -7517.278} C_VEL
LIN {X 0,Y 470.087,Z 420.3,A -85,B 0,C 180,E1 -7517.585,E2 -7517.585} C_VEL
LIN {X 0,Y 469.611,Z 432.834,A -85,B 0,C 180,E1 -7518.258,E2 -7518.258} C_VEL
LIN {X 0,Y 469.165,Z 444.236,A -85,B 0,C 180,E1 -7519.054,E2 -7519.054} C_VEL
LIN {X 0,Y 468.697,Z 454.497,A -85,B 0,C 180,E1 -7519.949,E2 -7519.949} C_VEL
LIN {X 0,Y 468.291,Z 463.609,A -85,B 0,C 180,E1 -7520.927,E2 -7520.927} C_VEL
LIN {X 0,Y 467.818,Z 473.286,A -85,B 0,C 180,E1 -7522.208,E2 -7522.208} C_VEL
LIN {X 0,Y 467.435,Z 481.524,A -85,B 0,C 180,E1 -7523.568,E2 -7523.568} C_VEL
LIN {X 0,Y 467.219,Z 487.152,A -85,B 0,C 180,E1 -7524.721,E2 -7524.721} C_VEL
LIN {X 0,Y 466.956,Z 492.731,A -85,B 0,C 180,E1 -7526.161,E2 -7526.161} C_VEL
LIN {X 0,Y 466.855,Z 496.562,A -85,B 0,C 180,E1 -7527.452,E2 -7527.452} C_VEL
LIN {X 0,Y 466.8,Z 498.313,A -85,B 0,C 180,E1 -7528.202,E2 -7528.202} C_VEL
LIN {X 0,Y 466.661,Z 500.172,A -85,B 0,C 180,E1 -7529.201,E2 -7529.201} C_VEL
LIN {X 0,Y 466.62,Z 501.988,A -85,B 0,C 180,E1 -7530.866,E2 -7530.866} C_VEL
LIN {X 0,Y 466.594,Z 502.312,A -85,B 0,C 180,E1 -7532.697,E2 -7532.697} C_VEL
LIN {X 0,Y 466.638,Z 501.331,A -85,B 0,C 180,E1 -7534.103,E2 -7534.103} C_VEL
LIN {X 0,Y 466.71,Z 500.022,A -85,B 0,C 180,E1 -7535.063,E2 -7535.063} C_VEL
LIN {X 0,Y 466.861,Z 496.736,A -85,B 0,C 180,E1 -7536.663,E2 -7536.663} C_VEL
LIN {X 0,Y 466.994,Z 493.127,A -85,B 0,C 180,E1 -7537.9,E2 -7537.9} C_VEL
LIN {X 0,Y 467.201,Z 487.77,A -85,B 0,C 180,E1 -7539.315,E2 -7539.315} C_VEL
LIN {X 0,Y 467.495,Z 481.072,A -85,B 0,C 180,E1 -7540.688,E2 -7540.688} C_VEL
LIN {X 0,Y 467.892,Z 472.581,A -85,B 0,C 180,E1 -7542.067,E2 -7542.067} C_VEL
LIN {X 0,Y 468.361,Z 463.838,A -85,B 0,C 180,E1 -7543.211,E2 -7543.211} C_VEL
LIN {X 0,Y 468.775,Z 454.767,A -85,B 0,C 180,E1 -7544.183,E2 -7544.183} C_VEL
LIN {X 0,Y 469.29,Z 443.71,A -85,B 0,C 180,E1 -7545.141,E2 -7545.141} C_VEL
LIN {X 0,Y 469.743,Z 432.248,A -85,B 0,C 180,E1 -7545.93,E2 -7545.93} C_VEL
LIN {X 0,Y 470.188,Z 420.34,A -85,B 0,C 180,E1 -7546.557,E2 -7546.557} C_VEL
LIN {X 0,Y 470.08,Z 413.502,A -85,B 0,C 180,E1 -7546.849,E2 -7546.849} C_VEL
LIN {X 0,Y 466.921,Z 400.414,A -85,B 0,C 180,E1 -7547.395,E2 -7547.395} C_VEL
LIN {X 0,Y 466.945,Z 397.268,A -85,B 0,C 180,E1 -7550.471,E2 -7550.471} C_VEL
LIN {X 0,Y 467.087,Z 394.513,A -85,B 0,C 180,E1 -7553.205,E2 -7553.205} C_VEL
LIN {X 0,Y 467.204,Z 392.058,A -85,B 0,C 180,E1 -7555.687,E2 -7555.687} C_VEL
LIN {X 0,Y 467.317,Z 388.688,A -85,B 0,C 180,E1 -7559.139,E2 -7559.139} C_VEL
LIN {X 0,Y 467.548,Z 387.012,A -85,B 0,C 180,E1 -7560.862,E2 -7560.862} C_VEL
LIN {X 0,Y 467.571,Z 382.951,A -85,B 0,C 180,E1 -7565.175,E2 -7565.175} C_VEL
LIN {X 0,Y 467.546,Z 382.25,A -85,B 0,C 180,E1 -7566.041,E2 -7566.041} C_VEL
LIN {X 0,Y 467.642,Z 382.238,A -85,B 0,C 180,E1 -7568.644,E2 -7568.644} C_VEL
LIN {X 0,Y 467.646,Z 382.234,A -85,B 0,C 180,E1 -7571.267,E2 -7571.267} C_VEL
LIN {X 0,Y 467.586,Z 382.241,A -85,B 0,C 180,E1 -7573.916,E2 -7573.916} C_VEL
LIN {X 0,Y 467.575,Z 382.243,A -85,B 0,C 180,E1 -7576.594,E2 -7576.594} C_VEL
LIN {X 0,Y 467.592,Z 382.243,A -85,B 0,C 180,E1 -7579.31,E2 -7579.31} C_VEL
LIN {X 0,Y 467.545,Z 382.249,A -85,B 0,C 180,E1 -7582.074,E2 -7582.074} C_VEL
LIN {X 0,Y 467.585,Z 382.241,A -85,B 0,C 180,E1 -7584.889,E2 -7584.889} C_VEL
LIN {X 0,Y 467.597,Z 382.24,A -85,B 0,C 180,E1 -7587.771,E2 -7587.771} C_VEL
LIN {X 0,Y 467.543,Z 382.247,A -85,B 0,C 180,E1 -7591.049,E2 -7591.049} C_VEL
LIN {X 0,Y 467.562,Z 382.245,A -85,B 0,C 180,E1 -7594.246,E2 -7594.246} C_VEL
LIN {X 0,Y 467.529,Z 382.25,A -85,B 0,C 180,E1 -7597.191,E2 -7597.191} C_VEL
LIN {X 0,Y 467.577,Z 382.245,A -85,B 0,C 180,E1 -7600.265,E2 -7600.265} C_VEL
LIN {X 0,Y 467.596,Z 382.242,A -85,B 0,C 180,E1 -7602.575,E2 -7602.575} C_VEL
LIN {X 0,Y 467.553,Z 382.247,A -85,B 0,C 180,E1 -7606.18,E2 -7606.18} C_VEL
LIN {X 0,Y 467.569,Z 382.352,A -85,B 0,C 180,E1 -7608.602,E2 -7608.602} C_VEL
LIN {X 0,Y 468.418,Z 387.135,A -85,B 0,C 180,E1 -7611.279,E2 -7611.279} C_VEL
LIN {X 0,Y 469.251,Z 392.472,A -85,B 0,C 180,E1 -7613.976,E2 -7613.976} C_VEL
LIN {X 0,Y 468.953,Z 397.76,A -85,B 0,C 180,E1 -7616.329,E2 -7616.329} C_VEL
LIN {X 0,Y 468.407,Z 404.961,A -85,B 0,C 180,E1 -7619.332,E2 -7619.332} C_VEL
LIN {X 0,Y 467.919,Z 413.884,A -85,B 0,C 180,E1 -7622.803,E2 -7622.803} C_VEL
LIN {X 0,Y 467.624,Z 421.415,A -85,B 0,C 180,E1 -7625.592,E2 -7625.592} C_VEL
LIN {X 0,Y 467.4,Z 429.239,A -85,B 0,C 180,E1 -7628.388,E2 -7628.388} C_VEL
LIN {X 0,Y 467.173,Z 438.465,A -85,B 0,C 180,E1 -7631.588,E2 -7631.588} C_VEL
LIN {X 0,Y 467.014,Z 447.273,A -85,B 0,C 180,E1 -7634.573,E2 -7634.573} C_VEL
LIN {X 0,Y 468.938,Z 462.208,A -85,B 0,C 180,E1 -7635.067,E2 -7635.067} C_VEL
LIN {X 0,Y 469.813,Z 470.757,A -85,B 0,C 180,E1 -7635.437,E2 -7635.437} C_VEL
LIN {X 0,Y 469.327,Z 482.566,A -85,B 0,C 180,E1 -7636.031,E2 -7636.031} C_VEL
LIN {X 0,Y 468.837,Z 494.091,A -85,B 0,C 180,E1 -7636.789,E2 -7636.789} C_VEL
LIN {X 0,Y 468.272,Z 505.386,A -85,B 0,C 180,E1 -7637.726,E2 -7637.726} C_VEL
LIN {X 0,Y 467.898,Z 515.296,A -85,B 0,C 180,E1 -7638.743,E2 -7638.743} C_VEL
LIN {X 0,Y 467.456,Z 523.968,A -85,B 0,C 180,E1 -7639.829,E2 -7639.829} C_VEL
LIN {X 0,Y 467.13,Z 532.418,A -85,B 0,C 180,E1 -7641.132,E2 -7641.132} C_VEL
LIN {X 0,Y 466.924,Z 539.245,A -85,B 0,C 180,E1 -7642.435,E2 -7642.435} C_VEL
LIN {X 0,Y 466.767,Z 545.509,A -85,B 0,C 180,E1 -7643.953,E2 -7643.953} C_VEL
LIN {X 0,Y 466.696,Z 549.58,A -85,B 0,C 180,E1 -7645.252,E2 -7645.252} C_VEL
LIN {X 0,Y 466.728,Z 552.597,A -85,B 0,C 180,E1 -7646.55,E2 -7646.55} C_VEL
LIN {X 0,Y 466.701,Z 554.036,A -85,B 0,C 180,E1 -7647.414,E2 -7647.414} C_VEL
LIN {X 0,Y 466.693,Z 555.067,A -85,B 0,C 180,E1 -7648.277,E2 -7648.277} C_VEL
LIN {X 0,Y 466.62,Z 555.699,A -85,B 0,C 180,E1 -7649.14,E2 -7649.14} C_VEL
LIN {X 0,Y 466.599,Z 555.933,A -85,B 0,C 180,E1 -7650.003,E2 -7650.003} C_VEL
LIN {X 0,Y 466.694,Z 555.127,A -85,B 0,C 180,E1 -7651.729,E2 -7651.729} C_VEL
LIN {X 0,Y 466.702,Z 554.129,A -85,B 0,C 180,E1 -7652.592,E2 -7652.592} C_VEL
LIN {X 0,Y 466.729,Z 552.717,A -85,B 0,C 180,E1 -7653.456,E2 -7653.456} C_VEL
LIN {X 0,Y 466.698,Z 549.746,A -85,B 0,C 180,E1 -7654.754,E2 -7654.754} C_VEL
LIN {X 0,Y 466.772,Z 545.72,A -85,B 0,C 180,E1 -7656.053,E2 -7656.053} C_VEL
LIN {X 0,Y 466.931,Z 539.515,A -85,B 0,C 180,E1 -7657.571,E2 -7657.571} C_VEL
LIN {X 0,Y 467.154,Z 532.746,A -85,B 0,C 180,E1 -7658.874,E2 -7658.874} C_VEL
LIN {X 0,Y 467.472,Z 524.349,A -85,B 0,C 180,E1 -7660.178,E2 -7660.178} C_VEL
